C07326=1174.282,254.736,-65.728,-177.284,7.391,148.606
C07327=1174.278,254.984,-65.755,-177.282,7.393,148.606
C07328=1174.274,255.233,-65.782,-177.279,7.396,148.606
C07329=1174.270,255.482,-65.809,-177.276,7.399,148.606
C07330=1174.265,255.729,-65.836,-177.274,7.401,148.606
C07331=1174.261,255.978,-65.863,-177.272,7.404,148.606
C07332=1174.256,256.226,-65.890,-177.268,7.407,148.606
C07333=1174.252,256.475,-65.919,-177.266,7.409,148.605
C07334=1174.248,256.723,-65.946,-177.263,7.412,148.605
C07335=1174.243,256.971,-65.973,-177.261,7.415,148.605
C07336=1174.238,257.221,-66.001,-177.258,7.417,148.605
C07337=1174.234,257.469,-66.029,-177.256,7.420,148.605
C07338=1174.229,257.717,-66.056,-177.253,7.423,148.605
C07339=1174.225,257.966,-66.083,-177.250,7.425,148.605
C07340=1174.221,258.214,-66.111,-177.248,7.428,148.605
C07341=1174.216,258.463,-66.139,-177.245,7.431,148.605
C07342=1174.212,258.711,-66.166,-177.242,7.434,148.605
C07343=1174.208,258.960,-66.194,-177.240,7.436,148.605
C07344=1174.204,259.208,-66.222,-177.237,7.439,148.604
C07345=1174.199,259.456,-66.249,-177.234,7.441,148.604
C07346=1174.195,259.705,-66.277,-177.232,7.444,148.604
C07347=1174.191,259.953,-66.304,-177.229,7.447,148.604
C07348=1174.186,260.201,-66.332,-177.226,7.450,148.604
C07349=1174.181,260.451,-66.360,-177.224,7.452,148.604
C07350=1174.177,260.699,-66.387,-177.221,7.455,148.604
C07351=1174.172,260.947,-66.414,-177.219,7.458,148.604
C07352=1174.169,261.196,-66.443,-177.216,7.461,148.604
C07353=1174.164,261.443,-66.470,-177.213,7.462,148.603
C07354=1174.160,261.692,-66.497,-177.211,7.465,148.603
C07355=1174.155,261.965,-66.528,-177.208,7.468,148.603
C07356=1174.150,262.239,-66.559,-177.205,7.471,148.603
C07357=1174.145,262.511,-66.589,-177.202,7.474,148.603
C07358=1174.140,262.785,-66.620,-177.200,7.477,148.603
C07359=1174.136,263.032,-66.648,-177.196,7.480,148.603
C07360=1174.132,263.281,-66.676,-177.194,7.483,148.603
C07361=1174.127,263.529,-66.704,-177.191,7.486,148.603
C07362=1174.123,263.778,-66.731,-177.189,7.488,148.603
C07363=1174.119,264.026,-66.759,-177.186,7.491,148.603
C07364=1174.114,264.274,-66.788,-177.183,7.494,148.603
C07365=1174.110,264.523,-66.816,-177.180,7.497,148.603
C07366=1174.105,264.772,-66.843,-177.178,7.499,148.602
C07367=1174.102,265.020,-66.871,-177.176,7.502,148.602
C07368=1174.096,265.268,-66.899,-177.173,7.505,148.602
C07369=1174.093,265.517,-66.927,-177.171,7.507,148.602
C07370=1174.088,265.765,-66.955,-177.168,7.510,148.602
C07371=1174.083,266.014,-66.983,-177.165,7.513,148.602
C07372=1174.079,266.262,-67.011,-177.162,7.516,148.602
C07373=1174.075,266.510,-67.039,-177.160,7.518,148.602
C07374=1174.070,266.759,-67.068,-177.157,7.521,148.602
C07375=1174.066,267.007,-67.095,-177.154,7.524,148.602
C07376=1174.062,267.255,-67.124,-177.152,7.527,148.602
C07377=1174.057,267.504,-67.152,-177.149,7.529,148.602
C07378=1174.053,267.752,-67.180,-177.147,7.532,148.602
C07379=1174.048,268.000,-67.208,-177.144,7.535,148.602
C07380=1174.045,268.249,-67.237,-177.141,7.538,148.601
C07381=1174.040,268.497,-67.264,-177.139,7.540,148.601
C07382=1174.036,268.746,-67.293,-177.136,7.543,148.601
C07383=1174.031,268.994,-67.321,-177.133,7.546,148.601
C07384=1174.027,269.242,-67.350,-177.131,7.549,148.601
C07385=1174.023,269.490,-67.377,-177.128,7.552,148.601
C07386=1174.018,269.739,-67.406,-177.126,7.554,148.601
C07387=1174.014,269.987,-67.434,-177.123,7.557,148.601
C07388=1174.009,270.236,-67.463,-177.120,7.560,148.601
C07389=1174.005,270.484,-67.490,-177.118,7.563,148.601
C07390=1174.000,270.733,-67.519,-177.115,7.565,148.601
C07391=1173.997,270.981,-67.547,-177.113,7.568,148.601
C07392=1173.992,271.229,-67.575,-177.110,7.571,148.601
C07393=1173.988,271.478,-67.604,-177.107,7.574,148.601
C07394=1173.983,271.726,-67.633,-177.104,7.577,148.601
C07395=1173.979,271.974,-67.661,-177.102,7.579,148.601
C07396=1173.974,272.222,-67.689,-177.100,7.582,148.601
C07397=1173.970,272.471,-67.718,-177.097,7.585,148.601
C07398=1173.966,272.720,-67.746,-177.094,7.588,148.600
C07399=1173.962,272.968,-67.774,-177.092,7.590,148.600
C07400=1173.957,273.216,-67.803,-177.089,7.593,148.600
C07401=1173.953,273.464,-67.831,-177.086,7.596,148.600
C07402=1173.949,273.713,-67.860,-177.084,7.599,148.600
C07403=1173.944,273.962,-67.889,-177.081,7.602,148.600
C07404=1173.940,274.209,-67.917,-177.079,7.604,148.600
C07405=1173.936,274.458,-67.946,-177.076,7.607,148.600
C07406=1173.931,274.706,-67.974,-177.073,7.610,148.600
C07407=1173.927,274.954,-68.003,-177.071,7.613,148.600
C07408=1173.923,275.203,-68.032,-177.068,7.616,148.600
C07409=1173.918,275.451,-68.060,-177.066,7.618,148.600
C07410=1173.914,275.699,-68.089,-177.063,7.621,148.600
C07411=1173.910,275.948,-68.117,-177.060,7.624,148.600
C07412=1173.905,276.196,-68.146,-177.057,7.627,148.600
C07413=1173.901,276.444,-68.175,-177.055,7.630,148.600
C07414=1173.897,276.693,-68.203,-177.052,7.632,148.600
C07415=1173.892,276.940,-68.232,-177.050,7.635,148.600
C07416=1173.888,277.189,-68.261,-177.047,7.638,148.600
C07417=1173.884,277.438,-68.290,-177.044,7.641,148.599
C07418=1173.880,277.686,-68.319,-177.041,7.644,148.599
C07419=1173.875,277.934,-68.347,-177.039,7.647,148.599
C07420=1173.871,278.182,-68.377,-177.037,7.650,148.600
C07421=1173.867,278.431,-68.405,-177.034,7.653,148.599
C07422=1173.862,278.678,-68.434,-177.032,7.656,148.599
C07423=1173.858,278.927,-68.462,-177.029,7.659,148.599
C07424=1173.854,279.176,-68.492,-177.026,7.662,148.599
C07425=1173.850,279.424,-68.520,-177.024,7.664,148.599
C07426=1173.845,279.672,-68.549,-177.021,7.667,148.599
C07427=1173.841,279.920,-68.579,-177.018,7.670,148.599
C07428=1173.836,280.169,-68.607,-177.016,7.673,148.599
C07429=1173.832,280.417,-68.637,-177.013,7.676,148.599
C07430=1173.828,280.665,-68.665,-177.010,7.679,148.599
C07431=1173.824,280.913,-68.694,-177.008,7.681,148.599
C07432=1173.820,281.162,-68.723,-177.005,7.684,148.599
C07433=1173.815,281.410,-68.752,-177.003,7.687,148.599
C07434=1173.810,281.658,-68.781,-177.000,7.690,148.599
C07435=1173.806,281.906,-68.811,-176.998,7.693,148.599
C07436=1173.802,282.155,-68.840,-176.995,7.696,148.599
C07437=1173.798,282.403,-68.868,-176.992,7.699,148.599
C07438=1173.794,282.651,-68.898,-176.990,7.701,148.599
C07439=1173.789,282.900,-68.926,-176.987,7.704,148.599
C07440=1173.785,283.148,-68.956,-176.984,7.707,148.599
C07441=1173.780,283.396,-68.985,-176.982,7.710,148.599
C07442=1173.776,283.644,-69.015,-176.979,7.713,148.599
C07443=1173.772,283.893,-69.044,-176.977,7.716,148.599
C07444=1173.767,284.141,-69.072,-176.975,7.718,148.599
C07445=1173.763,284.389,-69.102,-176.972,7.721,148.599
C07446=1173.759,284.637,-69.131,-176.969,7.724,148.599
C07447=1173.754,284.886,-69.161,-176.966,7.727,148.599
C07448=1173.750,285.134,-69.190,-176.964,7.730,148.599
C07449=1173.746,285.383,-69.219,-176.961,7.733,148.599
C07450=1173.741,285.630,-69.248,-176.959,7.737,148.599
C07451=1173.737,285.879,-69.277,-176.956,7.739,148.599
C07452=1173.733,286.127,-69.307,-176.954,7.742,148.599
C07453=1173.728,286.375,-69.336,-176.951,7.745,148.599
C07454=1173.724,286.623,-69.366,-176.948,7.748,148.599
C07455=1173.720,286.872,-69.395,-176.945,7.751,148.599
C07456=1173.716,287.120,-69.425,-176.943,7.754,148.599
C07457=1173.712,287.368,-69.454,-176.940,7.757,148.599
C07458=1173.707,287.616,-69.483,-176.938,7.760,148.599
C07459=1173.702,287.891,-69.516,-176.935,7.763,148.599
C07460=1173.698,288.166,-69.549,-176.932,7.766,148.599
C07461=1173.693,288.441,-69.581,-176.929,7.769,148.599
C07462=1173.688,288.715,-69.614,-176.926,7.773,148.599
C07463=1173.684,288.963,-69.644,-176.923,7.776,148.599
C07464=1173.680,289.212,-69.673,-176.921,7.779,148.599
C07465=1173.675,289.460,-69.703,-176.919,7.781,148.599
C07466=1173.671,289.708,-69.732,-176.916,7.784,148.599
C07467=1173.667,289.956,-69.761,-176.913,7.787,148.599
C07468=1173.663,290.205,-69.791,-176.911,7.790,148.599
C07469=1173.659,290.453,-69.820,-176.908,7.793,148.599
C07470=1173.654,290.702,-69.850,-176.905,7.796,148.599
C07471=1173.650,290.949,-69.881,-176.903,7.799,148.599
C07472=1173.646,291.197,-69.910,-176.900,7.802,148.599
C07473=1173.642,291.446,-69.939,-176.898,7.805,148.599
C07474=1173.637,291.694,-69.969,-176.895,7.807,148.599
C07475=1173.632,291.943,-69.999,-176.893,7.810,148.599
C07476=1173.629,292.190,-70.029,-176.890,7.814,148.599
C07477=1173.624,292.438,-70.059,-176.888,7.817,148.599
C07478=1173.620,292.687,-70.088,-176.885,7.820,148.599
C07479=1173.616,292.935,-70.117,-176.882,7.823,148.599
C07480=1173.611,293.183,-70.148,-176.879,7.826,148.599
C07481=1173.607,293.431,-70.178,-176.877,7.829,148.599
C07482=1173.603,293.680,-70.207,-176.874,7.832,148.599
C07483=1173.599,293.928,-70.237,-176.872,7.835,148.599
C07484=1173.594,294.176,-70.267,-176.869,7.837,148.599
C07485=1173.590,294.424,-70.297,-176.867,7.840,148.599
C07486=1173.586,294.672,-70.326,-176.864,7.843,148.599
C07487=1173.582,294.920,-70.356,-176.862,7.846,148.599
C07488=1173.577,295.169,-70.386,-176.859,7.849,148.599
C07489=1173.573,295.416,-70.417,-176.857,7.853,148.599
C07490=1173.569,295.664,-70.446,-176.854,7.856,148.599
C07491=1173.564,295.913,-70.476,-176.851,7.859,148.599
C07492=1173.560,296.161,-70.506,-176.849,7.862,148.599
C07493=1173.557,296.410,-70.536,-176.846,7.865,148.599
C07494=1173.552,296.658,-70.567,-176.844,7.868,148.599
C07495=1173.548,296.906,-70.596,-176.841,7.871,148.599
C07496=1173.543,297.154,-70.627,-176.839,7.873,148.599
C07497=1173.539,297.402,-70.657,-176.836,7.876,148.599
C07498=1173.535,297.650,-70.687,-176.834,7.879,148.599
C07499=1173.530,297.898,-70.717,-176.831,7.882,148.599
C07500=1173.526,298.146,-70.747,-176.828,7.885,148.599
C07501=1173.521,298.395,-70.777,-176.826,7.888,148.599
C07502=1173.518,298.642,-70.807,-176.823,7.891,148.599
C07503=1173.514,298.891,-70.838,-176.820,7.894,148.599
C07504=1173.509,299.139,-70.868,-176.818,7.897,148.599
C07505=1173.506,299.387,-70.898,-176.815,7.901,148.599
C07506=1173.501,299.635,-70.928,-176.813,7.904,148.599
C07507=1173.497,299.883,-70.958,-176.810,7.907,148.599
C07508=1173.492,300.131,-70.989,-176.807,7.910,148.599
C07509=1173.489,300.380,-71.019,-176.805,7.913,148.599
C07510=1173.484,300.628,-71.050,-176.802,7.916,148.599
C07511=1173.480,300.875,-71.080,-176.800,7.918,148.599
C07512=1173.475,301.124,-71.110,-176.798,7.921,148.600
C07513=1173.471,301.372,-71.140,-176.795,7.924,148.599
C07514=1173.467,301.620,-71.171,-176.792,7.927,148.599
C07515=1173.463,301.869,-71.200,-176.790,7.931,148.600
C07516=1173.458,302.117,-71.231,-176.787,7.934,148.600
C07517=1173.455,302.364,-71.261,-176.785,7.937,148.600
C07518=1173.450,302.612,-71.292,-176.782,7.940,148.600
C07519=1173.445,302.860,-71.323,-176.779,7.943,148.600
C07520=1173.442,303.109,-71.353,-176.777,7.946,148.600
C07521=1173.437,303.357,-71.384,-176.774,7.949,148.600
C07522=1173.433,303.605,-71.414,-176.772,7.952,148.600
C07523=1173.429,303.853,-71.444,-176.769,7.955,148.600
C07524=1173.424,304.101,-71.475,-176.766,7.958,148.600
C07525=1173.421,304.349,-71.506,-176.764,7.961,148.600
C07526=1173.416,304.598,-71.536,-176.761,7.964,148.600
C07527=1173.411,304.846,-71.567,-176.759,7.967,148.600
C07528=1173.407,305.093,-71.597,-176.756,7.971,148.600
C07529=1173.403,305.342,-71.628,-176.754,7.974,148.600
C07530=1173.399,305.590,-71.659,-176.751,7.977,148.600
C07531=1173.395,305.837,-71.689,-176.749,7.980,148.600
C07532=1173.391,306.086,-71.720,-176.746,7.983,148.600
C07533=1173.386,306.334,-71.751,-176.744,7.986,148.601
C07534=1173.382,306.582,-71.781,-176.741,7.988,148.600
C07535=1173.378,306.830,-71.812,-176.739,7.991,148.600
C07536=1173.374,307.078,-71.843,-176.736,7.995,148.601
C07537=1173.369,307.326,-71.874,-176.734,7.998,148.601
C07538=1173.365,307.574,-71.904,-176.731,8.001,148.601
C07539=1173.361,307.823,-71.935,-176.729,8.004,148.601
C07540=1173.357,308.071,-71.966,-176.726,8.007,148.601
C07541=1173.352,308.319,-71.996,-176.723,8.010,148.601
C07542=1173.349,308.567,-72.027,-176.721,8.013,148.601
C07543=1173.344,308.815,-72.058,-176.718,8.016,148.601
C07544=1173.340,309.062,-72.089,-176.716,8.020,148.601
C07545=1173.336,309.311,-72.120,-176.713,8.023,148.601
C07546=1173.331,309.559,-72.151,-176.710,8.025,148.601
C07547=1173.327,309.806,-72.181,-176.708,8.029,148.601
C07548=1173.323,310.055,-72.212,-176.705,8.032,148.601
C07549=1173.319,310.303,-72.243,-176.703,8.035,148.601
C07550=1173.314,310.550,-72.275,-176.700,8.038,148.601
C07551=1173.310,310.799,-72.306,-176.698,8.041,148.601
C07552=1173.306,311.047,-72.336,-176.695,8.044,148.602
C07553=1173.302,311.295,-72.367,-176.693,8.047,148.602
C07554=1173.298,311.543,-72.398,-176.690,8.051,148.602
C07555=1173.294,311.791,-72.429,-176.688,8.054,148.602
C07556=1173.290,312.039,-72.460,-176.685,8.057,148.602
C07557=1173.285,312.287,-72.491,-176.683,8.060,148.602
C07558=1173.281,312.535,-72.523,-176.680,8.063,148.602
C07559=1173.277,312.783,-72.554,-176.678,8.066,148.602
C07560=1173.272,313.031,-72.584,-176.675,8.069,148.602
C07561=1173.268,313.279,-72.616,-176.673,8.072,148.602
C07562=1173.264,313.527,-72.647,-176.670,8.075,148.602
C07563=1173.260,313.804,-72.682,-176.667,8.079,148.602
C07564=1173.254,314.081,-72.716,-176.664,8.083,148.602
C07565=1173.250,314.358,-72.751,-176.661,8.086,148.603
C07566=1173.245,314.634,-72.786,-176.659,8.090,148.603
C07567=1173.241,314.883,-72.817,-176.656,8.093,148.603
C07568=1173.237,315.130,-72.849,-176.653,8.096,148.603
C07569=1173.233,315.379,-72.880,-176.651,8.099,148.603
C07570=1173.229,315.626,-72.911,-176.648,8.102,148.603
C07571=1173.225,315.875,-72.943,-176.646,8.105,148.603
C07572=1173.220,316.122,-72.974,-176.643,8.108,148.603
C07573=1173.216,316.371,-73.005,-176.641,8.112,148.603
C07574=1173.212,316.618,-73.037,-176.638,8.115,148.603
C07575=1173.208,316.867,-73.068,-176.636,8.118,148.603
C07576=1173.204,317.114,-73.099,-176.633,8.121,148.603
C07577=1173.200,317.362,-73.131,-176.631,8.124,148.604
C07578=1173.195,317.610,-73.162,-176.628,8.127,148.604
C07579=1173.192,317.858,-73.194,-176.626,8.130,148.604
C07580=1173.187,318.106,-73.224,-176.623,8.133,148.604
C07581=1173.183,318.355,-73.257,-176.621,8.137,148.604
C07582=1173.178,318.602,-73.288,-176.618,8.140,148.604
C07583=1173.174,318.851,-73.319,-176.616,8.143,148.604
C07584=1173.170,319.099,-73.351,-176.613,8.147,148.604
C07585=1173.166,319.346,-73.383,-176.610,8.150,148.604
C07586=1173.162,319.595,-73.414,-176.608,8.153,148.604
C07587=1173.158,319.842,-73.445,-176.605,8.156,148.605
C07588=1173.153,320.091,-73.478,-176.603,8.159,148.605
C07589=1173.149,320.338,-73.509,-176.600,8.163,148.605
C07590=1173.145,320.587,-73.540,-176.598,8.166,148.605
C07591=1173.141,320.835,-73.572,-176.595,8.169,148.605
C07592=1173.137,321.082,-73.604,-176.593,8.172,148.605
C07593=1173.133,321.330,-73.636,-176.590,8.175,148.605
C07594=1173.128,321.578,-73.667,-176.588,8.178,148.605
C07595=1173.124,321.826,-73.699,-176.585,8.182,148.605
C07596=1173.121,322.074,-73.731,-176.583,8.185,148.606
C07597=1173.116,322.322,-73.762,-176.580,8.188,148.606
C07598=1173.112,322.570,-73.795,-176.578,8.191,148.606
C07599=1173.108,322.818,-73.826,-176.575,8.194,148.606
C07600=1173.104,323.066,-73.857,-176.573,8.197,148.606
C07601=1173.100,323.314,-73.889,-176.570,8.200,148.606
C07602=1173.095,323.562,-73.921,-176.568,8.204,148.606
C07603=1173.091,323.810,-73.953,-176.566,8.207,148.606
C07604=1173.087,324.058,-73.985,-176.563,8.210,148.606
C07605=1173.084,324.306,-74.017,-176.560,8.214,148.607
C07606=1173.079,324.553,-74.049,-176.557,8.217,148.607
C07607=1173.075,324.801,-74.081,-176.555,8.220,148.607
C07608=1173.071,325.049,-74.112,-176.552,8.223,148.607
C07609=1173.066,325.297,-74.145,-176.550,8.227,148.607
C07610=1173.062,325.545,-74.176,-176.548,8.230,148.607
C07611=1173.059,325.793,-74.208,-176.545,8.233,148.607
C07612=1173.054,326.041,-74.240,-176.543,8.236,148.607
C07613=1173.050,326.289,-74.272,-176.541,8.240,148.608
C07614=1173.046,326.537,-74.305,-176.538,8.243,148.608
C07615=1173.041,326.785,-74.336,-176.536,8.246,148.608
C07616=1173.038,327.033,-74.368,-176.533,8.249,148.608
C07617=1173.033,327.281,-74.400,-176.531,8.252,148.608
C07618=1173.030,327.528,-74.433,-176.528,8.255,148.608
C07619=1173.025,327.776,-74.465,-176.526,8.258,148.608
C07620=1173.021,328.024,-74.497,-176.523,8.263,148.608
C07621=1173.017,328.272,-74.529,-176.520,8.266,148.609
C07622=1173.013,328.520,-74.561,-176.518,8.269,148.609
C07623=1173.008,328.768,-74.593,-176.515,8.272,148.609
C07624=1173.004,329.016,-74.626,-176.513,8.275,148.609
C07625=1173.001,329.264,-74.658,-176.510,8.278,148.609
C07626=1172.996,329.512,-74.690,-176.508,8.282,148.609
C07627=1172.992,329.759,-74.721,-176.506,8.285,148.609
C07628=1172.988,330.007,-74.755,-176.503,8.288,148.609
C07629=1172.984,330.255,-74.786,-176.501,8.291,148.610
C07630=1172.980,330.503,-74.819,-176.499,8.295,148.610
C07631=1172.975,330.751,-74.850,-176.496,8.298,148.610
C07632=1172.971,330.998,-74.884,-176.493,8.302,148.610
C07633=1172.967,331.246,-74.915,-176.491,8.305,148.610
C07634=1172.963,331.495,-74.948,-176.488,8.308,148.610
C07635=1172.959,331.743,-74.981,-176.486,8.311,148.610
C07636=1172.955,331.990,-75.012,-176.483,8.315,148.611
C07637=1172.950,332.238,-75.045,-176.481,8.318,148.611
C07638=1172.947,332.486,-75.077,-176.478,8.321,148.611
C07639=1172.942,332.734,-75.110,-176.476,8.324,148.611
C07640=1172.938,332.982,-75.143,-176.474,8.328,148.611
C07641=1172.934,333.230,-75.175,-176.471,8.331,148.611
C07642=1172.930,333.478,-75.208,-176.468,8.335,148.612
C07643=1172.926,333.725,-75.240,-176.466,8.338,148.612
C07644=1172.922,333.973,-75.273,-176.464,8.341,148.612
C07645=1172.917,334.221,-75.305,-176.461,8.344,148.612
C07646=1172.914,334.468,-75.338,-176.459,8.348,148.612
C07647=1172.910,334.717,-75.370,-176.456,8.351,148.612
C07648=1172.905,334.964,-75.403,-176.454,8.354,148.613
C07649=1172.902,335.212,-75.435,-176.451,8.357,148.613
C07650=1172.897,335.459,-75.468,-176.449,8.360,148.613
C07651=1172.893,335.708,-75.500,-176.446,8.365,148.613
C07652=1172.889,335.955,-75.533,-176.444,8.368,148.613
C07653=1172.885,336.204,-75.565,-176.442,8.371,148.613
C07654=1172.881,336.451,-75.599,-176.439,8.374,148.613
C07655=1172.876,336.699,-75.632,-176.437,8.377,148.614
C07656=1172.873,336.947,-75.664,-176.434,8.381,148.614
C07657=1172.869,337.195,-75.697,-176.432,8.384,148.614
C07658=1172.864,337.443,-75.730,-176.430,8.387,148.614
C07659=1172.860,337.691,-75.762,-176.427,8.391,148.614
C07660=1172.857,337.938,-75.795,-176.424,8.394,148.615
C07661=1172.852,338.186,-75.828,-176.422,8.398,148.615
C07662=1172.848,338.434,-75.860,-176.420,8.401,148.615
C07663=1172.844,338.682,-75.894,-176.418,8.404,148.615
C07664=1172.840,338.930,-75.927,-176.415,8.408,148.615
C07665=1172.836,339.177,-75.959,-176.413,8.411,148.615
C07666=1172.831,339.425,-75.991,-176.410,8.415,148.616
C07667=1172.827,339.705,-76.029,-176.407,8.418,148.616
C07668=1172.822,339.984,-76.066,-176.405,8.422,148.616
C07669=1172.818,340.263,-76.103,-176.402,8.426,148.616
C07670=1172.813,340.542,-76.141,-176.399,8.430,148.617
C07671=1172.809,340.790,-76.174,-176.397,8.433,148.617
C07672=1172.805,341.038,-76.207,-176.394,8.436,148.617
C07673=1172.800,341.286,-76.239,-176.392,8.440,148.617
C07674=1172.796,341.534,-76.272,-176.389,8.443,148.617
C07675=1172.793,341.781,-76.305,-176.387,8.447,148.617
C07676=1172.789,342.029,-76.338,-176.385,8.450,148.618
C07677=1172.784,342.277,-76.371,-176.382,8.453,148.618
C07678=1172.780,342.524,-76.405,-176.380,8.457,148.618
C07679=1172.776,342.772,-76.438,-176.377,8.461,148.618
C07680=1172.772,343.020,-76.471,-176.375,8.464,148.619
C07681=1172.768,343.268,-76.504,-176.373,8.467,148.619
C07682=1172.764,343.515,-76.537,-176.370,8.471,148.619
C07683=1172.760,343.763,-76.570,-176.368,8.474,148.619
C07684=1172.756,344.011,-76.603,-176.366,8.477,148.619
C07685=1172.751,344.258,-76.637,-176.363,8.481,148.620
C07686=1172.747,344.506,-76.670,-176.360,8.484,148.620
C07687=1172.743,344.754,-76.703,-176.358,8.488,148.620
C07688=1172.740,345.002,-76.736,-176.356,8.491,148.620
C07689=1172.735,345.250,-76.770,-176.354,8.494,148.620
C07690=1172.731,345.498,-76.803,-176.351,8.498,148.621
C07691=1172.727,345.746,-76.836,-176.348,8.502,148.621
C07692=1172.723,345.993,-76.870,-176.346,8.505,148.621
C07693=1172.719,346.240,-76.903,-176.344,8.508,148.621
C07694=1172.714,346.488,-76.937,-176.342,8.512,148.621
C07695=1172.710,346.736,-76.970,-176.339,8.515,148.622
C07696=1172.706,346.984,-77.003,-176.337,8.519,148.622
C07697=1172.702,347.232,-77.036,-176.335,8.523,148.622
C07698=1172.699,347.479,-77.070,-176.332,8.526,148.623
C07699=1172.695,347.727,-77.104,-176.330,8.529,148.623
C07700=1172.690,347.975,-77.137,-176.328,8.533,148.623
C07701=1172.686,348.223,-77.170,-176.325,8.536,148.623
C07702=1172.682,348.470,-77.204,-176.323,8.540,148.623
C07703=1172.678,348.718,-77.237,-176.320,8.543,148.624
C07704=1172.674,348.966,-77.271,-176.318,8.547,148.624
C07705=1172.670,349.213,-77.305,-176.316,8.550,148.624
C07706=1172.666,349.461,-77.338,-176.313,8.553,148.624
C07707=1172.662,349.709,-77.371,-176.311,8.557,148.625
C07708=1172.658,349.956,-77.405,-176.308,8.561,148.625
C07709=1172.653,350.204,-77.439,-176.306,8.564,148.625
C07710=1172.650,350.452,-77.472,-176.304,8.568,148.625
C07711=1172.646,350.699,-77.506,-176.302,8.571,148.626
C07712=1172.642,350.947,-77.539,-176.299,8.575,148.626
C07713=1172.637,351.195,-77.573,-176.297,8.578,148.626
C07714=1172.633,351.442,-77.607,-176.295,8.582,148.626
C07715=1172.629,351.691,-77.640,-176.292,8.585,148.627
C07716=1172.626,351.938,-77.674,-176.290,8.588,148.627
C07717=1172.621,352.186,-77.708,-176.288,8.593,148.627
C07718=1172.617,352.433,-77.742,-176.285,8.596,148.627
C07719=1172.613,352.681,-77.776,-176.283,8.599,148.628
C07720=1172.610,352.929,-77.809,-176.281,8.603,148.628
C07721=1172.605,353.177,-77.843,-176.278,8.607,148.628
C07722=1172.601,353.424,-77.877,-176.276,8.610,148.629
C07723=1172.597,353.672,-77.911,-176.274,8.614,148.629
C07724=1172.593,353.920,-77.945,-176.271,8.617,148.629
C07725=1172.589,354.167,-77.979,-176.269,8.620,148.629
C07726=1172.585,354.414,-78.012,-176.267,8.625,148.630
C07727=1172.581,354.663,-78.047,-176.265,8.628,148.630
C07728=1172.577,354.910,-78.080,-176.262,8.631,148.630
C07729=1172.573,355.157,-78.114,-176.260,8.634,148.630
C07730=1172.569,355.405,-78.149,-176.258,8.639,148.631
C07731=1172.565,355.653,-78.182,-176.255,8.642,148.631
C07732=1172.560,355.901,-78.216,-176.253,8.646,148.631
C07733=1172.557,356.148,-78.251,-176.251,8.649,148.632
C07734=1172.553,356.396,-78.284,-176.248,8.653,148.632
C07735=1172.548,356.644,-78.318,-176.246,8.657,148.632
C07736=1172.545,356.891,-78.352,-176.244,8.660,148.632
C07737=1172.540,357.139,-78.387,-176.242,8.663,148.633
C07738=1172.536,357.387,-78.420,-176.239,8.668,148.633
C07739=1172.533,357.634,-78.454,-176.237,8.671,148.633
C07740=1172.528,357.882,-78.489,-176.235,8.675,148.634
C07741=1172.525,358.129,-78.523,-176.233,8.678,148.634
C07742=1172.520,358.378,-78.557,-176.230,8.682,148.634
C07743=1172.517,358.625,-78.591,-176.228,8.686,148.635
C07744=1172.512,358.872,-78.625,-176.226,8.689,148.635
C07745=1172.509,359.120,-78.659,-176.224,8.692,148.635
C07746=1172.504,359.367,-78.694,-176.221,8.697,148.636
C07747=1172.501,359.615,-78.728,-176.219,8.700,148.636
C07748=1172.496,359.863,-78.762,-176.217,8.704,148.636
C07749=1172.493,360.110,-78.796,-176.215,8.707,148.637
C07750=1172.488,360.358,-78.830,-176.212,8.711,148.637
C07751=1172.484,360.606,-78.864,-176.210,8.715,148.637
C07752=1172.480,360.854,-78.899,-176.208,8.718,148.638
C07753=1172.477,361.101,-78.933,-176.206,8.721,148.638
C07754=1172.472,361.348,-78.968,-176.203,8.726,148.638
C07755=1172.468,361.596,-79.002,-176.202,8.730,148.639
C07756=1172.464,361.843,-79.036,-176.199,8.733,148.639
C07757=1172.460,362.092,-79.071,-176.197,8.736,148.639
C07758=1172.456,362.339,-79.105,-176.195,8.741,148.640
C07759=1172.452,362.587,-79.140,-176.193,8.744,148.640
C07760=1172.448,362.834,-79.174,-176.191,8.748,148.641
C07761=1172.445,363.081,-79.209,-176.189,8.751,148.641
C07762=1172.440,363.329,-79.244,-176.187,8.755,148.641
C07763=1172.437,363.577,-79.278,-176.184,8.759,148.642
C07764=1172.433,363.824,-79.312,-176.182,8.762,148.642
C07765=1172.429,364.072,-79.347,-176.180,8.766,148.642
C07766=1172.425,364.319,-79.381,-176.178,8.770,148.643
C07767=1172.421,364.567,-79.416,-176.176,8.773,148.643
C07768=1172.416,364.815,-79.450,-176.174,8.777,148.643
C07769=1172.413,365.062,-79.485,-176.172,8.781,148.644
C07770=1172.409,365.309,-79.520,-176.170,8.785,148.644
C07771=1172.404,365.592,-79.560,-176.168,8.789,148.645
C07772=1172.399,365.874,-79.598,-176.166,8.793,148.645
C07773=1172.395,366.156,-79.638,-176.163,8.797,148.646
C07774=1172.390,366.438,-79.678,-176.161,8.801,148.646
C07775=1172.387,366.685,-79.713,-176.159,8.805,148.647
C07776=1172.383,366.933,-79.747,-176.157,8.809,148.647
C07777=1172.379,367.181,-79.782,-176.155,8.812,148.647
C07778=1172.374,367.428,-79.816,-176.154,8.816,148.648
C07779=1172.371,367.675,-79.851,-176.152,8.820,148.648
C07780=1172.367,367.923,-79.886,-176.150,8.823,148.649
C07781=1172.363,368.171,-79.921,-176.147,8.828,148.649
C07782=1172.358,368.418,-79.956,-176.146,8.831,148.650
C07783=1172.354,368.666,-79.991,-176.144,8.835,148.650
C07784=1172.351,368.913,-80.024,-176.142,8.838,148.651
C07785=1172.347,369.160,-80.060,-176.140,8.842,148.651
C07786=1172.343,369.409,-80.095,-176.139,8.846,148.652
C07787=1172.339,369.655,-80.130,-176.137,8.850,148.652
C07788=1172.335,369.904,-80.165,-176.135,8.853,148.652
C07789=1172.330,370.151,-80.199,-176.133,8.857,148.653
C07790=1172.326,370.398,-80.235,-176.132,8.861,148.653
C07791=1172.323,370.646,-80.269,-176.130,8.864,148.654
C07792=1172.319,370.893,-80.304,-176.128,8.868,148.654
C07793=1172.315,371.141,-80.339,-176.127,8.872,148.655
C07794=1172.311,371.388,-80.374,-176.125,8.875,148.655
C07795=1172.307,371.636,-80.409,-176.123,8.879,148.656
C07796=1172.303,371.884,-80.445,-176.122,8.883,148.656
C07797=1172.299,372.131,-80.479,-176.120,8.886,148.657
C07798=1172.295,372.378,-80.515,-176.119,8.890,148.657
C07799=1172.291,372.627,-80.550,-176.117,8.893,148.658
C07800=1172.287,372.873,-80.585,-176.116,8.897,148.659
C07801=1172.284,373.121,-80.620,-176.114,8.901,148.659
C07802=1172.279,373.368,-80.654,-176.112,8.905,148.660
C07803=1172.276,373.616,-80.690,-176.111,8.908,148.660
C07804=1172.272,373.864,-80.724,-176.110,8.911,148.661
C07805=1172.267,374.110,-80.760,-176.108,8.915,148.661
C07806=1172.264,374.358,-80.795,-176.106,8.919,148.662
C07807=1172.260,374.606,-80.830,-176.105,8.923,148.662
C07808=1172.255,374.853,-80.865,-176.104,8.927,148.663
C07809=1172.252,375.100,-80.901,-176.102,8.929,148.663
C07810=1172.248,375.348,-80.936,-176.101,8.933,148.664
C07811=1172.244,375.596,-80.971,-176.100,8.937,148.665
C07812=1172.240,375.843,-81.006,-176.099,8.940,148.665
C07813=1172.236,376.091,-81.041,-176.097,8.944,148.666
C07814=1172.232,376.338,-81.077,-176.095,8.948,148.666
C07815=1172.228,376.585,-81.112,-176.095,8.951,148.667
C07816=1172.224,376.833,-81.147,-176.093,8.955,148.667
C07817=1172.220,377.081,-81.182,-176.092,8.959,148.668
C07818=1172.216,377.328,-81.217,-176.091,8.962,148.669
C07819=1172.212,377.575,-81.254,-176.090,8.966,148.669
C07820=1172.208,377.823,-81.289,-176.089,8.969,148.670
C07821=1172.204,378.071,-81.324,-176.087,8.973,148.670
C07822=1172.200,378.318,-81.359,-176.086,8.976,148.671
C07823=1172.196,378.565,-81.395,-176.085,8.980,148.672
C07824=1172.192,378.813,-81.430,-176.084,8.984,148.672
C07825=1172.188,379.060,-81.465,-176.083,8.987,148.673
C07826=1172.184,379.308,-81.500,-176.082,8.990,148.673
C07827=1172.181,379.555,-81.536,-176.081,8.994,148.674
C07828=1172.177,379.803,-81.571,-176.080,8.997,148.675
C07829=1172.172,380.050,-81.607,-176.079,9.001,148.675
C07830=1172.168,380.297,-81.643,-176.078,9.004,148.676
C07831=1172.165,380.545,-81.678,-176.077,9.007,148.677
C07832=1172.161,380.792,-81.714,-176.076,9.012,148.677
C07833=1172.156,381.040,-81.748,-176.075,9.015,148.678
C07834=1172.153,381.287,-81.784,-176.074,9.018,148.679
C07835=1172.149,381.535,-81.819,-176.073,9.022,148.679
C07836=1172.145,381.783,-81.856,-176.073,9.025,148.680
C07837=1172.141,382.030,-81.891,-176.072,9.028,148.681
C07838=1172.137,382.277,-81.926,-176.071,9.032,148.681
C07839=1172.133,382.524,-81.962,-176.070,9.035,148.682
C07840=1172.129,382.772,-81.997,-176.069,9.039,148.683
C07841=1172.126,383.019,-82.033,-176.069,9.042,148.683
C07842=1172.121,383.267,-82.069,-176.068,9.045,148.684
C07843=1172.117,383.514,-82.104,-176.067,9.048,148.685
C07844=1172.113,383.762,-82.140,-176.067,9.051,148.685
C07845=1172.110,384.009,-82.175,-176.066,9.055,148.686
C07846=1172.106,384.257,-82.211,-176.065,9.058,148.687
C07847=1172.101,384.504,-82.247,-176.064,9.062,148.687
C07848=1172.097,384.751,-82.282,-176.063,9.065,148.688
C07849=1172.094,384.999,-82.318,-176.063,9.069,148.689
C07850=1172.090,385.246,-82.353,-176.063,9.071,148.690
C07851=1172.086,385.494,-82.389,-176.062,9.074,148.690
C07852=1172.082,385.741,-82.425,-176.062,9.078,148.691
C07853=1172.078,385.988,-82.460,-176.061,9.081,148.691
C07854=1172.074,386.236,-82.496,-176.061,9.084,148.692
C07855=1172.070,386.484,-82.532,-176.060,9.088,148.693
C07856=1172.066,386.730,-82.568,-176.059,9.091,148.694
C07857=1172.063,386.978,-82.604,-176.060,9.093,148.694
C07858=1172.059,387.225,-82.639,-176.059,9.097,148.695
C07859=1172.054,387.473,-82.675,-176.059,9.100,148.696
C07860=1172.050,387.720,-82.711,-176.058,9.103,148.696
C07861=1172.047,387.968,-82.746,-176.058,9.106,148.697
C07862=1172.043,388.215,-82.782,-176.058,9.109,148.698
C07863=1172.039,388.463,-82.818,-176.057,9.112,148.699
C07864=1172.035,388.710,-82.854,-176.057,9.115,148.699
C07865=1172.031,388.957,-82.889,-176.057,9.118,148.700
C07866=1172.027,389.204,-82.925,-176.057,9.121,148.701
C07867=1172.023,389.452,-82.961,-176.056,9.124,148.701
C07868=1172.019,389.699,-82.996,-176.056,9.127,148.702
C07869=1172.015,389.947,-83.033,-176.056,9.130,148.703
C07870=1172.011,390.194,-83.069,-176.056,9.133,148.704
C07871=1172.008,390.442,-83.104,-176.056,9.136,148.704
C07872=1172.004,390.689,-83.140,-176.056,9.139,148.705
C07873=1171.999,390.936,-83.176,-176.056,9.142,148.706
C07874=1171.995,391.184,-83.211,-176.055,9.144,148.706
C07875=1171.991,391.468,-83.253,-176.055,9.148,148.707
C07876=1171.986,391.753,-83.294,-176.055,9.151,148.708
C07877=1171.983,392.038,-83.336,-176.055,9.154,148.709
C07878=1171.978,392.323,-83.377,-176.055,9.158,148.710
C07879=1171.974,392.571,-83.413,-176.055,9.160,148.711
C07880=1171.970,392.817,-83.449,-176.055,9.163,148.711
C07881=1171.966,393.064,-83.484,-176.055,9.166,148.712
C07882=1171.962,393.312,-83.520,-176.055,9.169,148.713
C07883=1171.958,393.560,-83.556,-176.055,9.171,148.714
C07884=1171.955,393.807,-83.592,-176.055,9.174,148.714
C07885=1171.950,394.054,-83.628,-176.055,9.176,148.715
C07886=1171.946,394.302,-83.664,-176.055,9.179,148.715
C07887=1171.943,394.549,-83.699,-176.055,9.181,148.716
C07888=1171.939,394.797,-83.736,-176.055,9.185,148.717
C07889=1171.935,395.044,-83.772,-176.055,9.187,148.718
C07890=1171.930,395.291,-83.808,-176.055,9.190,148.718
C07891=1171.927,395.538,-83.844,-176.056,9.192,148.719
C07892=1171.923,395.786,-83.879,-176.056,9.195,148.720
C07893=1171.919,396.033,-83.915,-176.056,9.197,148.721
C07894=1171.915,396.281,-83.951,-176.056,9.200,148.721
C07895=1171.911,396.528,-83.988,-176.056,9.203,148.722
C07896=1171.907,396.776,-84.023,-176.056,9.205,148.723
C07897=1171.904,397.023,-84.059,-176.056,9.208,148.723
C07898=1171.899,397.270,-84.096,-176.057,9.210,148.724
C07899=1171.896,397.518,-84.131,-176.057,9.212,148.725
C07900=1171.891,397.766,-84.168,-176.057,9.215,148.725
C07901=1171.887,398.012,-84.203,-176.058,9.217,148.726
C07902=1171.884,398.259,-84.239,-176.057,9.219,148.727
C07903=1171.879,398.507,-84.275,-176.057,9.222,148.727
C07904=1171.876,398.754,-84.311,-176.058,9.225,148.728
C07905=1171.872,399.002,-84.348,-176.058,9.227,148.729
C07906=1171.868,399.249,-84.383,-176.059,9.229,148.729
C07907=1171.864,399.496,-84.420,-176.059,9.231,148.730
C07908=1171.860,399.744,-84.455,-176.059,9.234,148.731
C07909=1171.857,399.991,-84.492,-176.059,9.237,148.732
C07910=1171.852,400.239,-84.528,-176.060,9.238,148.732
C07911=1171.849,400.486,-84.563,-176.060,9.241,148.733
C07912=1171.845,400.733,-84.600,-176.060,9.243,148.734
C07913=1171.841,400.981,-84.636,-176.060,9.246,148.734
C07914=1171.836,401.228,-84.672,-176.060,9.247,148.735
C07915=1171.833,401.475,-84.708,-176.061,9.250,148.736
C07916=1171.828,401.723,-84.744,-176.061,9.253,148.736
C07917=1171.825,401.970,-84.780,-176.061,9.254,148.737
C07918=1171.821,402.217,-84.816,-176.061,9.257,148.737
C07919=1171.817,402.465,-84.852,-176.061,9.259,148.738
C07920=1171.813,402.712,-84.888,-176.062,9.261,148.739
C07921=1171.809,402.960,-84.924,-176.062,9.263,148.740
C07922=1171.806,403.206,-84.961,-176.062,9.266,148.740
C07923=1171.801,403.454,-84.997,-176.063,9.267,148.741
C07924=1171.798,403.702,-85.032,-176.063,9.270,148.741
C07925=1171.794,403.949,-85.069,-176.063,9.272,148.742
C07926=1171.790,404.196,-85.105,-176.064,9.274,148.743
C07927=1171.786,404.444,-85.142,-176.064,9.276,148.743
C07928=1171.782,404.691,-85.177,-176.064,9.278,148.744
C07929=1171.778,404.939,-85.213,-176.065,9.280,148.745
C07930=1171.774,405.186,-85.250,-176.065,9.283,148.745
C07931=1171.771,405.433,-85.285,-176.065,9.285,148.746
C07932=1171.766,405.680,-85.322,-176.065,9.287,148.747
C07933=1171.762,405.927,-85.357,-176.066,9.289,148.747
C07934=1171.758,406.174,-85.394,-176.066,9.291,148.748
C07935=1171.755,406.422,-85.430,-176.066,9.293,148.748
C07936=1171.750,406.670,-85.466,-176.067,9.295,148.749
C07937=1171.747,406.917,-85.502,-176.067,9.297,148.750
C07938=1171.742,407.164,-85.538,-176.067,9.299,148.750
C07939=1171.739,407.411,-85.574,-176.068,9.301,148.751
C07940=1171.735,407.659,-85.611,-176.068,9.303,148.751
C07941=1171.731,407.906,-85.647,-176.068,9.305,148.752
C07942=1171.727,408.154,-85.683,-176.068,9.307,148.753
C07943=1171.724,408.401,-85.719,-176.069,9.309,148.753
C07944=1171.719,408.649,-85.755,-176.069,9.311,148.754
C07945=1171.716,408.895,-85.792,-176.069,9.313,148.754
C07946=1171.711,409.143,-85.828,-176.070,9.315,148.755
C07947=1171.708,409.390,-85.864,-176.070,9.317,148.756
C07948=1171.704,409.638,-85.900,-176.070,9.319,148.756
C07949=1171.700,409.885,-85.936,-176.070,9.321,148.757
C07950=1171.696,410.133,-85.973,-176.071,9.323,148.757
C07951=1171.693,410.379,-86.009,-176.071,9.324,148.758
C07952=1171.688,410.627,-86.045,-176.071,9.327,148.759
C07953=1171.685,410.874,-86.081,-176.072,9.328,148.759
C07954=1171.680,411.122,-86.117,-176.072,9.330,148.760
C07955=1171.677,411.370,-86.153,-176.072,9.332,148.760
C07956=1171.673,411.617,-86.190,-176.073,9.334,148.761
C07957=1171.669,411.864,-86.225,-176.073,9.336,148.762
C07958=1171.665,412.111,-86.262,-176.073,9.338,148.762
C07959=1171.661,412.359,-86.298,-176.074,9.339,148.763
C07960=1171.657,412.606,-86.335,-176.073,9.342,148.763
C07961=1171.654,412.853,-86.371,-176.074,9.343,148.764
C07962=1171.649,413.101,-86.407,-176.074,9.345,148.764
C07963=1171.646,413.348,-86.443,-176.074,9.347,148.765
C07964=1171.642,413.595,-86.479,-176.075,9.349,148.765
C07965=1171.638,413.842,-86.516,-176.075,9.350,148.766
C07966=1171.634,414.090,-86.552,-176.075,9.353,148.767
C07967=1171.630,414.337,-86.588,-176.076,9.354,148.767
C07968=1171.626,414.585,-86.624,-176.076,9.356,148.767
C07969=1171.621,414.831,-86.661,-176.077,9.358,148.768
C07970=1171.618,415.079,-86.696,-176.076,9.360,148.769
C07971=1171.614,415.327,-86.733,-176.077,9.362,148.769
C07972=1171.611,415.574,-86.769,-176.077,9.363,148.770
C07973=1171.609,415.821,-86.805,-176.077,9.365,148.770
C07974=1171.607,416.069,-86.841,-176.077,9.367,148.771
C07975=1171.606,416.344,-86.881,-176.078,9.368,148.771
C07976=1171.607,416.619,-86.921,-176.078,9.371,148.772
C07977=1171.609,416.895,-86.961,-176.078,9.372,148.772
C07978=1171.612,417.169,-87.000,-176.079,9.374,148.773
C07979=1171.191,417.170,-87.045,-176.082,9.385,148.777
C07980=1171.188,416.892,-87.005,-176.081,9.383,148.776
C07981=1171.185,416.614,-86.965,-176.081,9.382,148.776
C07982=1171.185,416.336,-86.924,-176.081,9.379,148.775
C07983=1171.185,416.057,-86.884,-176.081,9.378,148.775
C07984=1171.187,415.810,-86.847,-176.080,9.376,148.774
C07985=1171.189,415.563,-86.811,-176.080,9.374,148.773
C07986=1171.193,415.315,-86.776,-176.080,9.372,148.773
C07987=1171.197,415.068,-86.739,-176.080,9.371,148.772
C07988=1171.201,414.821,-86.704,-176.079,9.369,148.772
C07989=1171.205,414.573,-86.667,-176.079,9.367,148.771
C07990=1171.209,414.326,-86.631,-176.079,9.365,148.771
C07991=1171.213,414.079,-86.594,-176.078,9.364,148.770
C07992=1171.217,413.831,-86.558,-176.078,9.361,148.770
C07993=1171.220,413.584,-86.522,-176.078,9.360,148.769
C07994=1171.224,413.337,-86.485,-176.077,9.358,148.769
C07995=1171.228,413.089,-86.449,-176.077,9.356,148.768
C07996=1171.232,412.842,-86.413,-176.077,9.354,148.767
C07997=1171.236,412.595,-86.377,-176.077,9.353,148.767
C07998=1171.240,412.347,-86.340,-176.077,9.350,148.766
C07999=1171.244,412.100,-86.305,-176.076,9.349,148.766
C08000=1171.248,411.853,-86.268,-176.076,9.347,148.765
C08001=1171.251,411.605,-86.232,-176.076,9.345,148.765
C08002=1171.255,411.358,-86.195,-176.075,9.343,148.764
C08003=1171.259,411.110,-86.160,-176.075,9.342,148.763
C08004=1171.263,410.863,-86.123,-176.075,9.339,148.763
C08005=1171.267,410.616,-86.087,-176.074,9.338,148.762
C08006=1171.271,410.369,-86.051,-176.074,9.336,148.762
C08007=1171.275,410.121,-86.015,-176.074,9.334,148.761
C08008=1171.279,409.874,-85.978,-176.073,9.332,148.761
C08009=1171.282,409.626,-85.943,-176.073,9.329,148.760
C08010=1171.286,409.379,-85.906,-176.073,9.328,148.759
C08011=1171.291,409.131,-85.870,-176.072,9.326,148.759
C08012=1171.294,408.885,-85.833,-176.072,9.324,148.758
C08013=1171.299,408.637,-85.797,-176.072,9.322,148.758
C08014=1171.302,408.390,-85.761,-176.072,9.319,148.757
C08015=1171.306,408.142,-85.725,-176.071,9.318,148.756
C08016=1171.310,407.895,-85.689,-176.071,9.316,148.756
C08017=1171.313,407.648,-85.653,-176.071,9.314,148.755
C08018=1171.318,407.400,-85.616,-176.070,9.312,148.755
C08019=1171.321,407.153,-85.581,-176.070,9.310,148.754
C08020=1171.326,406.905,-85.544,-176.070,9.308,148.753
C08021=1171.330,406.659,-85.509,-176.070,9.306,148.753
C08022=1171.334,406.411,-85.472,-176.069,9.304,148.752
C08023=1171.337,406.164,-85.436,-176.069,9.302,148.751
C08024=1171.342,405.916,-85.400,-176.068,9.300,148.751
C08025=1171.345,405.670,-85.364,-176.068,9.297,148.750
C08026=1171.349,405.422,-85.328,-176.068,9.296,148.749
C08027=1171.353,405.175,-85.291,-176.068,9.293,148.749
C08028=1171.357,404.927,-85.255,-176.067,9.292,148.748
C08029=1171.361,404.680,-85.220,-176.067,9.289,148.748
C08030=1171.365,404.432,-85.183,-176.066,9.287,148.747
C08031=1171.369,404.185,-85.147,-176.067,9.285,148.746
C08032=1171.373,403.938,-85.110,-176.066,9.283,148.746
C08033=1171.376,403.690,-85.075,-176.066,9.281,148.745
C08034=1171.380,403.443,-85.038,-176.065,9.279,148.744
C08035=1171.384,403.196,-85.002,-176.065,9.277,148.744
C08036=1171.389,402.948,-84.966,-176.065,9.274,148.743
C08037=1171.392,402.701,-84.930,-176.064,9.272,148.743
C08038=1171.396,402.453,-84.894,-176.064,9.270,148.742
C08039=1171.400,402.206,-84.858,-176.063,9.268,148.741
C08040=1171.403,401.959,-84.822,-176.063,9.266,148.740
C08041=1171.407,401.711,-84.785,-176.064,9.263,148.740
C08042=1171.411,401.464,-84.750,-176.063,9.262,148.739
C08043=1171.416,401.217,-84.714,-176.063,9.259,148.739
C08044=1171.419,400.970,-84.678,-176.063,9.256,148.738
C08045=1171.424,400.722,-84.641,-176.062,9.255,148.737
C08046=1171.428,400.475,-84.606,-176.062,9.252,148.736
C08047=1171.432,400.227,-84.569,-176.062,9.250,148.736
C08048=1171.435,399.980,-84.533,-176.061,9.247,148.735
C08049=1171.439,399.733,-84.497,-176.061,9.246,148.735
C08050=1171.443,399.485,-84.461,-176.061,9.243,148.734
C08051=1171.447,399.238,-84.426,-176.061,9.240,148.733
C08052=1171.451,398.991,-84.389,-176.061,9.238,148.732
C08053=1171.454,398.743,-84.353,-176.060,9.236,148.732
C08054=1171.459,398.495,-84.317,-176.060,9.233,148.731
C08055=1171.462,398.248,-84.281,-176.060,9.231,148.730
C08056=1171.466,398.001,-84.245,-176.060,9.228,148.730
C08057=1171.471,397.754,-84.209,-176.059,9.226,148.729
C08058=1171.474,397.507,-84.173,-176.059,9.223,148.728
C08059=1171.479,397.259,-84.137,-176.059,9.221,148.727
C08060=1171.482,397.012,-84.101,-176.059,9.218,148.727
C08061=1171.486,396.765,-84.065,-176.058,9.216,148.726
C08062=1171.490,396.517,-84.029,-176.058,9.214,148.725
C08063=1171.494,396.269,-83.993,-176.058,9.211,148.725
C08064=1171.498,396.022,-83.957,-176.058,9.209,148.724
C08065=1171.501,395.775,-83.921,-176.058,9.206,148.723
C08066=1171.506,395.527,-83.885,-176.058,9.204,148.723
C08067=1171.509,395.280,-83.849,-176.058,9.201,148.722
C08068=1171.513,395.033,-83.813,-176.058,9.199,148.721
C08069=1171.518,394.785,-83.777,-176.057,9.196,148.721
C08070=1171.521,394.539,-83.741,-176.058,9.193,148.720
C08071=1171.525,394.291,-83.706,-176.058,9.190,148.719
C08072=1171.529,394.043,-83.669,-176.058,9.188,148.718
C08073=1171.533,393.796,-83.634,-176.057,9.185,148.718
C08074=1171.537,393.549,-83.597,-176.057,9.182,148.717
C08075=1171.541,393.301,-83.561,-176.057,9.180,148.716
C08076=1171.544,393.054,-83.526,-176.057,9.177,148.716
C08077=1171.549,392.806,-83.490,-176.057,9.174,148.715
C08078=1171.553,392.560,-83.454,-176.057,9.171,148.714
C08079=1171.556,392.312,-83.418,-176.057,9.169,148.713
C08080=1171.561,392.026,-83.377,-176.057,9.165,148.713
C08081=1171.565,391.742,-83.335,-176.057,9.163,148.712
C08082=1171.570,391.457,-83.294,-176.057,9.159,148.711
C08083=1171.575,391.172,-83.252,-176.057,9.155,148.710
C08084=1171.578,390.925,-83.217,-176.057,9.153,148.709
C08085=1171.582,390.677,-83.181,-176.058,9.150,148.709
C08086=1171.586,390.430,-83.145,-176.058,9.147,148.708
C08087=1171.590,390.183,-83.109,-176.058,9.145,148.707
C08088=1171.594,389.936,-83.074,-176.058,9.141,148.706
C08089=1171.598,389.688,-83.038,-176.058,9.139,148.706
C08090=1171.602,389.441,-83.002,-176.058,9.135,148.705
C08091=1171.606,389.193,-82.966,-176.059,9.132,148.704
C08092=1171.609,388.946,-82.930,-176.059,9.129,148.703
C08093=1171.613,388.698,-82.894,-176.059,9.126,148.703
C08094=1171.617,388.451,-82.859,-176.059,9.124,148.702
C08095=1171.621,388.204,-82.823,-176.060,9.120,148.701
C08096=1171.626,387.956,-82.787,-176.060,9.117,148.701
C08097=1171.629,387.709,-82.752,-176.060,9.114,148.700
C08098=1171.633,387.462,-82.715,-176.060,9.111,148.699
C08099=1171.636,387.214,-82.680,-176.061,9.108,148.699
C08100=1171.641,386.967,-82.644,-176.061,9.105,148.698
C08101=1171.645,386.720,-82.609,-176.061,9.102,148.697
C08102=1171.649,386.472,-82.573,-176.062,9.098,148.696
C08103=1171.653,386.225,-82.537,-176.063,9.095,148.696
C08104=1171.657,385.977,-82.501,-176.063,9.092,148.695
C08105=1171.661,385.730,-82.466,-176.063,9.089,148.694
C08106=1171.664,385.482,-82.430,-176.064,9.086,148.694
C08107=1171.669,385.235,-82.394,-176.064,9.083,148.693
C08108=1171.673,384.987,-82.359,-176.065,9.080,148.692
C08109=1171.676,384.741,-82.323,-176.065,9.076,148.691
C08110=1171.680,384.493,-82.287,-176.066,9.073,148.691
C08111=1171.684,384.246,-82.252,-176.067,9.070,148.690
C08112=1171.688,383.998,-82.215,-176.068,9.066,148.689
C08113=1171.692,383.751,-82.180,-176.069,9.063,148.689
C08114=1171.696,383.503,-82.145,-176.069,9.059,148.688
C08115=1171.700,383.256,-82.109,-176.070,9.056,148.687
C08116=1171.704,383.008,-82.073,-176.070,9.053,148.687
C08117=1171.708,382.761,-82.037,-176.071,9.050,148.686
C08118=1171.712,382.514,-82.002,-176.071,9.046,148.685
C08119=1171.716,382.266,-81.967,-176.073,9.042,148.685
C08120=1171.719,382.019,-81.931,-176.073,9.039,148.684
C08121=1171.723,381.771,-81.896,-176.074,9.036,148.683
C08122=1171.728,381.524,-81.861,-176.075,9.033,148.683
C08123=1171.732,381.276,-81.825,-176.076,9.029,148.682
C08124=1171.735,381.029,-81.789,-176.077,9.026,148.681
C08125=1171.739,380.781,-81.754,-176.078,9.022,148.681
C08126=1171.743,380.534,-81.718,-176.079,9.019,148.680
C08127=1171.747,380.287,-81.683,-176.079,9.015,148.679
C08128=1171.751,380.039,-81.647,-176.080,9.012,148.679
C08129=1171.755,379.791,-81.611,-176.082,9.008,148.678
C08130=1171.759,379.544,-81.576,-176.083,9.005,148.678
C08131=1171.763,379.297,-81.541,-176.084,9.001,148.677
C08132=1171.767,379.049,-81.506,-176.084,8.998,148.676
C08133=1171.771,378.802,-81.470,-176.086,8.994,148.675
C08134=1171.774,378.554,-81.435,-176.087,8.991,148.675
C08135=1171.779,378.307,-81.400,-176.088,8.987,148.674
C08136=1171.783,378.059,-81.363,-176.089,8.984,148.674
C08137=1171.787,377.811,-81.329,-176.090,8.980,148.673
C08138=1171.791,377.565,-81.293,-176.091,8.977,148.673
C08139=1171.795,377.317,-81.258,-176.093,8.973,148.672
C08140=1171.799,377.070,-81.222,-176.094,8.969,148.671
C08141=1171.802,376.822,-81.187,-176.095,8.966,148.671
C08142=1171.807,376.575,-81.152,-176.096,8.962,148.670
C08143=1171.810,376.327,-81.117,-176.097,8.959,148.670
C08144=1171.814,376.080,-81.081,-176.099,8.955,148.669
C08145=1171.818,375.833,-81.046,-176.100,8.951,148.668
C08146=1171.822,375.585,-81.011,-176.102,8.947,148.668
C08147=1171.826,375.337,-80.976,-176.103,8.944,148.667
C08148=1171.830,375.090,-80.940,-176.104,8.941,148.667
C08149=1171.834,374.842,-80.906,-176.106,8.937,148.666
C08150=1171.838,374.595,-80.870,-176.107,8.933,148.666
C08151=1171.842,374.347,-80.835,-176.108,8.930,148.665
C08152=1171.846,374.100,-80.800,-176.110,8.926,148.665
C08153=1171.850,373.852,-80.765,-176.111,8.922,148.664
C08154=1171.853,373.605,-80.729,-176.113,8.919,148.663
C08155=1171.858,373.357,-80.695,-176.115,8.915,148.663
C08156=1171.862,373.110,-80.659,-176.115,8.912,148.662
C08157=1171.866,372.863,-80.625,-176.117,8.908,148.662
C08158=1171.870,372.615,-80.589,-176.119,8.904,148.661
C08159=1171.874,372.367,-80.554,-176.120,8.901,148.661
C08160=1171.878,372.120,-80.519,-176.122,8.897,148.660
C08161=1171.882,371.873,-80.483,-176.124,8.893,148.660
C08162=1171.885,371.625,-80.449,-176.126,8.889,148.659
C08163=1171.889,371.378,-80.414,-176.127,8.885,148.659
C08164=1171.893,371.130,-80.379,-176.129,8.882,148.658
C08165=1171.897,370.882,-80.344,-176.130,8.878,148.658
C08166=1171.902,370.635,-80.309,-176.132,8.874,148.657
C08167=1171.905,370.387,-80.274,-176.134,8.871,148.657
C08168=1171.910,370.140,-80.239,-176.136,8.867,148.656
C08169=1171.914,369.892,-80.204,-176.137,8.863,148.656
C08170=1171.917,369.644,-80.169,-176.139,8.860,148.655
C08171=1171.921,369.397,-80.135,-176.141,8.856,148.655
C08172=1171.925,369.150,-80.099,-176.143,8.852,148.654
C08173=1171.929,368.902,-80.065,-176.145,8.849,148.654
C08174=1171.933,368.654,-80.030,-176.146,8.845,148.653
C08175=1171.938,368.407,-79.995,-176.148,8.841,148.653
C08176=1171.941,368.160,-79.961,-176.150,8.838,148.652
C08177=1171.945,367.912,-79.925,-176.151,8.834,148.652
C08178=1171.949,367.665,-79.891,-176.153,8.830,148.652
C08179=1171.953,367.417,-79.856,-176.155,8.827,148.651
C08180=1171.958,367.169,-79.821,-176.158,8.822,148.651
C08181=1171.961,366.922,-79.786,-176.159,8.819,148.650
C08182=1171.965,366.675,-79.752,-176.161,8.815,148.650
C08183=1171.969,366.426,-79.717,-176.163,8.812,148.649
C08184=1171.974,366.145,-79.678,-176.166,8.807,148.649
C08185=1171.978,365.862,-79.638,-176.167,8.804,148.649
C08186=1171.983,365.581,-79.598,-176.170,8.799,148.648
C08187=1171.987,365.298,-79.559,-176.172,8.795,148.648
C08188=1171.991,365.051,-79.525,-176.174,8.791,148.647
C08189=1171.995,364.803,-79.490,-176.176,8.788,148.647
C08190=1172.000,364.556,-79.455,-176.178,8.784,148.646
C08191=1172.003,364.309,-79.420,-176.181,8.780,148.646
C08192=1172.007,364.061,-79.386,-176.182,8.776,148.646
C08193=1172.011,363.813,-79.351,-176.185,8.773,148.645
C08194=1172.015,363.566,-79.317,-176.187,8.769,148.645
C08195=1172.019,363.318,-79.282,-176.188,8.766,148.644
C08196=1172.023,363.071,-79.249,-176.191,8.761,148.644
C08197=1172.027,362.823,-79.214,-176.193,8.758,148.644
C08198=1172.031,362.575,-79.179,-176.195,8.754,148.643
C08199=1172.035,362.327,-79.145,-176.197,8.751,148.643
C08200=1172.039,362.080,-79.111,-176.200,8.747,148.643
C08201=1172.043,361.832,-79.076,-176.201,8.743,148.642
C08202=1172.047,361.585,-79.041,-176.204,8.740,148.642
C08203=1172.051,361.338,-79.007,-176.206,8.736,148.642
C08204=1172.055,361.090,-78.972,-176.208,8.732,148.641
C08205=1172.059,360.842,-78.939,-176.210,8.728,148.641
C08206=1172.063,360.594,-78.904,-176.213,8.725,148.641
C08207=1172.067,360.347,-78.870,-176.214,8.721,148.640
C08208=1172.070,360.099,-78.836,-176.217,8.717,148.640
C08209=1172.075,359.852,-78.801,-176.219,8.714,148.640
C08210=1172.080,359.604,-78.767,-176.221,8.710,148.639
C08211=1172.083,359.356,-78.733,-176.224,8.707,148.639
C08212=1172.087,359.109,-78.698,-176.226,8.703,148.639
C08213=1172.091,358.861,-78.664,-176.228,8.699,148.638
C08214=1172.095,358.614,-78.629,-176.230,8.696,148.638
C08215=1172.099,358.366,-78.596,-176.232,8.692,148.638
C08216=1172.103,358.118,-78.562,-176.235,8.688,148.637
C08217=1172.107,357.871,-78.527,-176.237,8.685,148.637
C08218=1172.111,357.624,-78.494,-176.239,8.681,148.637
C08219=1172.115,357.376,-78.459,-176.242,8.678,148.637
C08220=1172.119,357.128,-78.426,-176.244,8.674,148.636
C08221=1172.124,356.880,-78.391,-176.246,8.670,148.636
C08222=1172.127,356.633,-78.357,-176.249,8.667,148.636
C08223=1172.131,356.385,-78.322,-176.251,8.663,148.635
C08224=1172.136,356.137,-78.289,-176.253,8.659,148.635
C08225=1172.139,355.890,-78.255,-176.256,8.656,148.635
C08226=1172.143,355.642,-78.221,-176.258,8.652,148.634
C08227=1172.148,355.395,-78.187,-176.260,8.648,148.634
C08228=1172.152,355.146,-78.153,-176.263,8.645,148.634
C08229=1172.155,354.899,-78.119,-176.265,8.642,148.634
C08230=1172.159,354.652,-78.086,-176.267,8.638,148.633
C08231=1172.163,354.403,-78.051,-176.269,8.635,148.633
C08232=1172.167,354.156,-78.017,-176.272,8.631,148.633
C08233=1172.171,353.909,-77.984,-176.274,8.627,148.633
C08234=1172.176,353.661,-77.949,-176.276,8.624,148.632
C08235=1172.180,353.413,-77.916,-176.278,8.620,148.632
C08236=1172.183,353.166,-77.882,-176.281,8.616,148.632
C08237=1172.188,352.918,-77.848,-176.283,8.613,148.631
C08238=1172.191,352.670,-77.814,-176.286,8.610,148.631
C08239=1172.196,352.422,-77.781,-176.288,8.606,148.631
C08240=1172.199,352.175,-77.747,-176.290,8.602,148.630
C08241=1172.204,351.927,-77.713,-176.293,8.599,148.630
C08242=1172.208,351.680,-77.679,-176.295,8.595,148.630
C08243=1172.212,351.431,-77.646,-176.297,8.592,148.630
C08244=1172.216,351.184,-77.612,-176.300,8.589,148.630
C08245=1172.220,350.936,-77.578,-176.302,8.584,148.629
C08246=1172.224,350.689,-77.544,-176.304,8.581,148.629
C08247=1172.228,350.441,-77.511,-176.306,8.578,148.629
C08248=1172.232,350.193,-77.478,-176.309,8.574,148.628
C08249=1172.236,349.946,-77.443,-176.312,8.570,148.628
C08250=1172.241,349.698,-77.410,-176.314,8.567,148.628
C08251=1172.244,349.451,-77.376,-176.316,8.564,148.628
C08252=1172.248,349.202,-77.343,-176.318,8.560,148.628
C08253=1172.252,348.955,-77.309,-176.321,8.557,148.627
C08254=1172.256,348.707,-77.276,-176.323,8.553,148.627
C08255=1172.261,348.459,-77.242,-176.325,8.549,148.627
C08256=1172.265,348.212,-77.209,-176.328,8.546,148.626
C08257=1172.269,347.964,-77.175,-176.330,8.543,148.626
C08258=1172.273,347.717,-77.142,-176.332,8.539,148.626
C08259=1172.276,347.468,-77.108,-176.335,8.535,148.626
C08260=1172.281,347.221,-77.075,-176.337,8.532,148.626
C08261=1172.285,346.973,-77.042,-176.340,8.529,148.625
C08262=1172.289,346.725,-77.009,-176.342,8.525,148.625
C08263=1172.293,346.478,-76.974,-176.344,8.522,148.625
C08264=1172.298,346.230,-76.941,-176.347,8.518,148.625
C08265=1172.302,345.982,-76.908,-176.349,8.515,148.624
C08266=1172.306,345.735,-76.875,-176.352,8.511,148.624
C08267=1172.309,345.486,-76.841,-176.354,8.508,148.624
C08268=1172.314,345.238,-76.808,-176.356,8.505,148.624
C08269=1172.318,344.991,-76.775,-176.358,8.501,148.624
C08270=1172.322,344.743,-76.742,-176.361,8.497,148.623
C08271=1172.326,344.496,-76.708,-176.364,8.494,148.623
C08272=1172.330,344.248,-76.675,-176.366,8.491,148.623
C08273=1172.334,344.000,-76.641,-176.368,8.487,148.623
C08274=1172.338,343.753,-76.608,-176.370,8.484,148.622
C08275=1172.342,343.505,-76.575,-176.373,8.481,148.622
C08276=1172.346,343.257,-76.542,-176.376,8.477,148.622
C08277=1172.350,343.010,-76.509,-176.378,8.473,148.622
C08278=1172.355,342.762,-76.476,-176.380,8.470,148.622
C08279=1172.359,342.514,-76.443,-176.382,8.467,148.621
C08280=1172.363,342.266,-76.409,-176.385,8.463,148.621
C08281=1172.367,342.018,-76.377,-176.387,8.460,148.621
C08282=1172.371,341.770,-76.344,-176.390,8.456,148.621
C08283=1172.376,341.523,-76.311,-176.393,8.453,148.621
C08284=1172.380,341.275,-76.277,-176.395,8.450,148.620
C08285=1172.384,341.027,-76.244,-176.397,8.446,148.620
C08286=1172.387,340.780,-76.212,-176.399,8.443,148.620
C08287=1172.391,340.532,-76.179,-176.402,8.440,148.620
C08288=1172.396,340.252,-76.141,-176.405,8.436,148.620
C08289=1172.401,339.973,-76.104,-176.407,8.432,148.619
C08290=1172.405,339.694,-76.068,-176.410,8.429,148.619
C08291=1172.410,339.414,-76.030,-176.413,8.424,148.619
C08292=1172.414,339.166,-75.997,-176.415,8.421,148.619
C08293=1172.418,338.919,-75.964,-176.418,8.418,148.619
C08294=1172.422,338.671,-75.931,-176.420,8.414,148.618
C08295=1172.426,338.423,-75.899,-176.423,8.410,148.618
C08296=1172.430,338.175,-75.866,-176.425,8.407,148.618
C08297=1172.434,337.927,-75.833,-176.428,8.404,148.618
C08298=1172.439,337.679,-75.800,-176.430,8.401,148.618
C08299=1172.443,337.431,-75.767,-176.432,8.398,148.618
C08300=1172.446,337.184,-75.734,-176.434,8.394,148.617
C08301=1172.451,336.937,-75.702,-176.437,8.391,148.617
C08302=1172.456,336.688,-75.669,-176.440,8.387,148.617
C08303=1172.459,336.441,-75.637,-176.442,8.384,148.617
C08304=1172.463,336.193,-75.604,-176.445,8.381,148.617
C08305=1172.468,335.945,-75.571,-176.447,8.377,148.616
C08306=1172.472,335.697,-75.538,-176.449,8.374,148.616
C08307=1172.475,335.449,-75.506,-176.452,8.371,148.616
C08308=1172.480,335.201,-75.473,-176.454,8.368,148.616
C08309=1172.484,334.953,-75.440,-176.456,8.364,148.616
C08310=1172.487,334.706,-75.408,-176.459,8.360,148.616
C08311=1172.492,334.457,-75.375,-176.462,8.357,148.616
C08312=1172.497,334.210,-75.343,-176.464,8.354,148.615
C08313=1172.500,333.962,-75.311,-176.467,8.351,148.615
C08314=1172.504,333.715,-75.278,-176.469,8.347,148.615
C08315=1172.509,333.466,-75.245,-176.472,8.344,148.615
C08316=1172.512,333.219,-75.213,-176.474,8.341,148.615
C08317=1172.517,332.970,-75.180,-176.476,8.338,148.615
C08318=1172.521,332.723,-75.147,-176.479,8.334,148.614
C08319=1172.525,332.475,-75.116,-176.482,8.331,148.614
C08320=1172.530,332.227,-75.083,-176.484,8.327,148.614
C08321=1172.533,331.980,-75.051,-176.486,8.324,148.614
C08322=1172.537,331.731,-75.018,-176.489,8.321,148.614
C08323=1172.541,331.484,-74.986,-176.491,8.318,148.614
C08324=1172.546,331.236,-74.953,-176.494,8.314,148.613
C08325=1172.550,330.988,-74.921,-176.496,8.311,148.613
C08326=1172.554,330.740,-74.888,-176.499,8.308,148.613
C08327=1172.558,330.492,-74.856,-176.501,8.305,148.613
C08328=1172.562,330.244,-74.824,-176.504,8.301,148.613
C08329=1172.567,329.996,-74.792,-176.506,8.298,148.613
C08330=1172.570,329.749,-74.760,-176.509,8.294,148.613
C08331=1172.575,329.501,-74.727,-176.511,8.291,148.612
C08332=1172.578,329.253,-74.695,-176.514,8.288,148.612
C08333=1172.583,329.005,-74.663,-176.516,8.285,148.612
C08334=1172.587,328.757,-74.631,-176.518,8.282,148.612
C08335=1172.591,328.509,-74.598,-176.521,8.279,148.612
C08336=1172.595,328.261,-74.566,-176.523,8.275,148.612
C08337=1172.600,328.013,-74.534,-176.526,8.272,148.612
C08338=1172.604,327.765,-74.502,-176.528,8.269,148.612
C08339=1172.607,327.518,-74.470,-176.531,8.265,148.611
C08340=1172.612,327.270,-74.437,-176.533,8.261,148.611
C08341=1172.616,327.022,-74.406,-176.536,8.259,148.611
C08342=1172.620,326.774,-74.373,-176.538,8.255,148.611
C08343=1172.624,326.526,-74.342,-176.541,8.252,148.611
C08344=1172.628,326.278,-74.310,-176.543,8.249,148.611
C08345=1172.633,326.030,-74.278,-176.546,8.246,148.611
C08346=1172.637,325.782,-74.246,-176.548,8.243,148.611
C08347=1172.641,325.534,-74.213,-176.551,8.239,148.610
C08348=1172.645,325.286,-74.182,-176.553,8.236,148.610
C08349=1172.649,325.038,-74.150,-176.556,8.233,148.610
C08350=1172.653,324.790,-74.118,-176.558,8.230,148.610
C08351=1172.658,324.543,-74.086,-176.561,8.227,148.610
C08352=1172.661,324.295,-74.054,-176.563,8.223,148.610
C08353=1172.666,324.046,-74.022,-176.566,8.219,148.610
C08354=1172.670,323.799,-73.990,-176.569,8.216,148.610
C08355=1172.674,323.551,-73.959,-176.571,8.213,148.609
C08356=1172.678,323.303,-73.927,-176.574,8.210,148.609
C08357=1172.683,323.055,-73.895,-176.576,8.207,148.609
C08358=1172.686,322.807,-73.863,-176.578,8.203,148.609
C08359=1172.690,322.559,-73.831,-176.581,8.200,148.609
C08360=1172.695,322.311,-73.800,-176.583,8.197,148.609
C08361=1172.699,322.063,-73.768,-176.586,8.194,148.609
C08362=1172.703,321.815,-73.736,-176.588,8.191,148.609
C08363=1172.707,321.568,-73.704,-176.591,8.188,148.609
C08364=1172.711,321.319,-73.673,-176.593,8.185,148.608
C08365=1172.715,321.072,-73.641,-176.596,8.182,148.608
C08366=1172.720,320.823,-73.609,-176.598,8.178,148.608
C08367=1172.724,320.575,-73.578,-176.601,8.175,148.608
C08368=1172.728,320.328,-73.546,-176.603,8.172,148.608
C08369=1172.732,320.080,-73.514,-176.605,8.169,148.608
C08370=1172.736,319.832,-73.483,-176.608,8.166,148.608
C08371=1172.741,319.583,-73.451,-176.611,8.162,148.608
C08372=1172.744,319.335,-73.419,-176.614,8.159,148.608
C08373=1172.749,319.087,-73.388,-176.616,8.155,148.607
C08374=1172.753,318.839,-73.357,-176.619,8.152,148.607
C08375=1172.757,318.592,-73.325,-176.621,8.149,148.607
C08376=1172.761,318.343,-73.294,-176.624,8.146,148.607
C08377=1172.765,318.096,-73.262,-176.626,8.143,148.607
C08378=1172.769,317.848,-73.231,-176.629,8.140,148.607
C08379=1172.774,317.600,-73.200,-176.631,8.136,148.607
C08380=1172.778,317.352,-73.167,-176.634,8.133,148.607
C08381=1172.782,317.104,-73.136,-176.636,8.130,148.607
C08382=1172.786,316.856,-73.105,-176.639,8.127,148.607
C08383=1172.791,316.608,-73.073,-176.641,8.124,148.606
C08384=1172.795,316.360,-73.042,-176.644,8.121,148.606
C08385=1172.799,316.112,-73.011,-176.646,8.118,148.606
C08386=1172.803,315.864,-72.980,-176.649,8.115,148.606
C08387=1172.807,315.616,-72.948,-176.651,8.111,148.606
C08388=1172.811,315.368,-72.917,-176.654,8.108,148.606
C08389=1172.816,315.120,-72.885,-176.657,8.105,148.606
C08390=1172.820,314.872,-72.854,-176.659,8.102,148.606
C08391=1172.824,314.624,-72.823,-176.662,8.099,148.606
C08392=1172.829,314.347,-72.789,-176.664,8.095,148.606
C08393=1172.833,314.070,-72.754,-176.667,8.092,148.606
C08394=1172.838,313.794,-72.718,-176.670,8.088,148.605
C08395=1172.842,313.516,-72.683,-176.673,8.085,148.605
C08396=1172.847,313.269,-72.653,-176.676,8.082,148.605
C08397=1172.851,313.021,-72.622,-176.678,8.079,148.605
C08398=1172.855,312.773,-72.590,-176.681,8.076,148.605
C08399=1172.859,312.525,-72.559,-176.683,8.072,148.605
C08400=1172.863,312.276,-72.528,-176.686,8.069,148.605
C08401=1172.868,312.029,-72.497,-176.688,8.066,148.605
C08402=1172.872,311.781,-72.466,-176.691,8.063,148.605
C08403=1172.876,311.532,-72.435,-176.693,8.060,148.605
C08404=1172.880,311.284,-72.405,-176.696,8.057,148.605
C08405=1172.884,311.036,-72.373,-176.698,8.054,148.605
C08406=1172.889,310.788,-72.342,-176.701,8.050,148.605
C08407=1172.893,310.540,-72.311,-176.703,8.047,148.605
C08408=1172.897,310.292,-72.280,-176.706,8.044,148.605
C08409=1172.902,310.044,-72.249,-176.708,8.041,148.604
C08410=1172.906,309.796,-72.218,-176.711,8.038,148.604
C08411=1172.909,309.548,-72.187,-176.713,8.035,148.604
C08412=1172.914,309.300,-72.157,-176.716,8.032,148.604
C08413=1172.918,309.051,-72.125,-176.719,8.029,148.604
C08414=1172.923,308.803,-72.095,-176.721,8.026,148.604
C08415=1172.927,308.555,-72.064,-176.724,8.023,148.604
C08416=1172.931,308.307,-72.033,-176.726,8.019,148.604
C08417=1172.935,308.060,-72.002,-176.729,8.016,148.604
C08418=1172.939,307.812,-71.971,-176.732,8.013,148.604
C08419=1172.943,307.563,-71.940,-176.734,8.010,148.604
C08420=1172.947,307.316,-71.910,-176.737,8.007,148.604
C08421=1172.952,307.068,-71.879,-176.739,8.004,148.604
C08422=1172.957,306.820,-71.848,-176.742,8.001,148.604
C08423=1172.961,306.571,-71.817,-176.744,7.998,148.604
C08424=1172.964,306.323,-71.787,-176.747,7.995,148.603
C08425=1172.969,306.075,-71.756,-176.749,7.992,148.603
C08426=1172.973,305.827,-71.725,-176.752,7.989,148.604
C08427=1172.977,305.579,-71.695,-176.754,7.985,148.603
C08428=1172.982,305.331,-71.664,-176.757,7.982,148.603
C08429=1172.986,305.083,-71.633,-176.760,7.979,148.603
C08430=1172.990,304.834,-71.604,-176.762,7.976,148.603
C08431=1172.994,304.586,-71.573,-176.765,7.973,148.603
C08432=1172.999,304.338,-71.542,-176.768,7.970,148.603
C08433=1173.003,304.091,-71.512,-176.770,7.967,148.603
C08434=1173.007,303.842,-71.481,-176.773,7.964,148.603
C08435=1173.012,303.594,-71.450,-176.775,7.961,148.603
C08436=1173.015,303.346,-71.420,-176.777,7.958,148.603
C08437=1173.020,303.098,-71.389,-176.780,7.955,148.603
C08438=1173.024,302.849,-71.359,-176.782,7.952,148.603
C08439=1173.028,302.601,-71.329,-176.785,7.949,148.603
C08440=1173.033,302.354,-71.298,-176.787,7.946,148.603
C08441=1173.037,302.106,-71.268,-176.790,7.943,148.603
C08442=1173.042,301.857,-71.238,-176.792,7.940,148.603
C08443=1173.045,301.609,-71.207,-176.795,7.937,148.603
C08444=1173.050,301.361,-71.176,-176.798,7.934,148.603
C08445=1173.053,301.113,-71.146,-176.800,7.931,148.603
C08446=1173.058,300.865,-71.116,-176.803,7.928,148.603
C08447=1173.062,300.617,-71.086,-176.806,7.925,148.603
C08448=1173.067,300.369,-71.055,-176.808,7.922,148.603
C08449=1173.070,300.120,-71.025,-176.811,7.918,148.602
C08450=1173.075,299.872,-70.995,-176.813,7.915,148.602
C08451=1173.079,299.625,-70.964,-176.816,7.912,148.602
C08452=1173.084,299.376,-70.934,-176.818,7.909,148.602
C08453=1173.088,299.128,-70.904,-176.821,7.906,148.602
C08454=1173.093,298.880,-70.874,-176.824,7.903,148.602
C08455=1173.096,298.632,-70.844,-176.827,7.900,148.602
C08456=1173.100,298.383,-70.813,-176.828,7.898,148.602
C08457=1173.105,298.135,-70.783,-176.831,7.895,148.602
C08458=1173.109,297.888,-70.753,-176.834,7.892,148.602
C08459=1173.113,297.639,-70.723,-176.836,7.888,148.602
C08460=1173.117,297.391,-70.693,-176.839,7.885,148.602
C08461=1173.122,297.143,-70.663,-176.842,7.882,148.602
C08462=1173.126,296.895,-70.633,-176.844,7.879,148.602
C08463=1173.130,296.647,-70.603,-176.847,7.876,148.602
C08464=1173.135,296.399,-70.573,-176.849,7.873,148.602
C08465=1173.138,296.150,-70.543,-176.852,7.870,148.602
C08466=1173.142,295.902,-70.513,-176.855,7.867,148.602
C08467=1173.147,295.654,-70.482,-176.857,7.864,148.602
C08468=1173.151,295.405,-70.453,-176.860,7.861,148.602
C08469=1173.155,295.158,-70.423,-176.862,7.859,148.602
C08470=1173.160,294.909,-70.393,-176.865,7.856,148.602
C08471=1173.164,294.662,-70.363,-176.867,7.852,148.602
C08472=1173.168,294.413,-70.333,-176.870,7.849,148.602
C08473=1173.173,294.165,-70.303,-176.872,7.846,148.602
C08474=1173.177,293.917,-70.273,-176.875,7.844,148.602
C08475=1173.181,293.669,-70.244,-176.878,7.841,148.602
C08476=1173.185,293.421,-70.214,-176.880,7.837,148.602
C08477=1173.190,293.173,-70.183,-176.883,7.834,148.602
C08478=1173.194,292.924,-70.154,-176.886,7.831,148.602
C08479=1173.198,292.676,-70.124,-176.888,7.828,148.602
C08480=1173.203,292.428,-70.095,-176.891,7.825,148.602
C08481=1173.207,292.180,-70.064,-176.893,7.823,148.602
C08482=1173.211,291.932,-70.035,-176.896,7.820,148.602
C08483=1173.216,291.683,-70.005,-176.898,7.817,148.602
C08484=1173.220,291.435,-69.976,-176.901,7.814,148.602
C08485=1173.224,291.187,-69.946,-176.903,7.811,148.602
C08486=1173.228,290.939,-69.916,-176.906,7.808,148.602
C08487=1173.233,290.690,-69.886,-176.909,7.805,148.602
C08488=1173.237,290.442,-69.857,-176.912,7.802,148.602
C08489=1173.241,290.194,-69.827,-176.914,7.799,148.602
C08490=1173.245,289.946,-69.798,-176.917,7.795,148.602
C08491=1173.249,289.697,-69.768,-176.919,7.793,148.602
C08492=1173.254,289.449,-69.739,-176.922,7.790,148.602
C08493=1173.258,289.201,-69.709,-176.924,7.787,148.602
C08494=1173.262,288.953,-69.679,-176.927,7.784,148.602
C08495=1173.267,288.705,-69.649,-176.930,7.781,148.602
C08496=1173.271,288.430,-69.618,-176.932,7.778,148.602
C08497=1173.276,288.156,-69.584,-176.935,7.774,148.602
C08498=1173.281,287.880,-69.552,-176.938,7.771,148.602
C08499=1173.285,287.605,-69.520,-176.941,7.768,148.602
C08500=1173.290,287.357,-69.490,-176.944,7.765,148.602
C08501=1173.295,287.109,-69.461,-176.946,7.762,148.602
C08502=1173.299,286.861,-69.431,-176.949,7.759,148.602
C08503=1173.303,286.612,-69.402,-176.952,7.756,148.602
C08504=1173.307,286.364,-69.372,-176.954,7.753,148.602
C08505=1173.312,286.116,-69.343,-176.956,7.751,148.602
C08506=1173.316,285.868,-69.313,-176.959,7.748,148.602
C08507=1173.320,285.619,-69.284,-176.962,7.745,148.602
C08508=1173.324,285.371,-69.254,-176.964,7.742,148.602
C08509=1173.329,285.124,-69.225,-176.967,7.739,148.602
C08510=1173.333,284.875,-69.196,-176.970,7.736,148.602
C08511=1173.338,284.626,-69.167,-176.972,7.733,148.602
C08512=1173.342,284.378,-69.138,-176.974,7.731,148.602
C08513=1173.346,284.130,-69.108,-176.977,7.728,148.602
C08514=1173.349,283.882,-69.079,-176.980,7.725,148.602
C08515=1173.354,283.634,-69.050,-176.983,7.722,148.602
C08516=1173.359,283.385,-69.021,-176.985,7.719,148.602
C08517=1173.363,283.137,-68.992,-176.988,7.716,148.602
C08518=1173.367,282.889,-68.963,-176.991,7.713,148.602
C08519=1173.371,282.641,-68.933,-176.992,7.710,148.602
C08520=1173.376,282.392,-68.905,-176.995,7.707,148.602
C08521=1173.381,282.144,-68.875,-176.998,7.704,148.602
C08522=1173.385,281.896,-68.846,-177.001,7.701,148.602
C08523=1173.389,281.647,-68.817,-177.003,7.698,148.602
C08524=1173.393,281.399,-68.788,-177.006,7.695,148.602
C08525=1173.397,281.151,-68.759,-177.009,7.692,148.602
C08526=1173.402,280.903,-68.730,-177.011,7.690,148.602
C08527=1173.406,280.654,-68.701,-177.014,7.687,148.602
C08528=1173.410,280.406,-68.671,-177.017,7.684,148.602
C08529=1173.415,280.158,-68.643,-177.019,7.681,148.602
C08530=1173.419,279.910,-68.614,-177.022,7.678,148.602
C08531=1173.423,279.661,-68.586,-177.024,7.675,148.602
C08532=1173.427,279.413,-68.556,-177.026,7.673,148.602
C08533=1173.432,279.165,-68.527,-177.029,7.670,148.602
C08534=1173.436,278.917,-68.499,-177.032,7.667,148.602
C08535=1173.440,278.668,-68.469,-177.035,7.664,148.602
C08536=1173.445,278.419,-68.441,-177.037,7.661,148.602
C08537=1173.449,278.172,-68.412,-177.040,7.658,148.603
C08538=1173.453,277.923,-68.383,-177.042,7.656,148.603
C08539=1173.457,277.675,-68.354,-177.045,7.653,148.603
C08540=1173.462,277.427,-68.326,-177.048,7.650,148.603
C08541=1173.467,277.179,-68.296,-177.051,7.647,148.603
C08542=1173.470,276.930,-68.268,-177.053,7.644,148.603
C08543=1173.476,276.682,-68.240,-177.055,7.642,148.603
C08544=1173.480,276.434,-68.210,-177.058,7.639,148.603
C08545=1173.483,276.185,-68.182,-177.061,7.636,148.603
C08546=1173.488,275.937,-68.153,-177.063,7.633,148.603
C08547=1173.493,275.689,-68.124,-177.066,7.630,148.603
C08548=1173.496,275.440,-68.096,-177.069,7.627,148.603
C08549=1173.501,275.192,-68.067,-177.071,7.625,148.603
C08550=1173.506,274.943,-68.038,-177.074,7.622,148.603
C08551=1173.509,274.695,-68.010,-177.076,7.619,148.603
C08552=1173.514,274.447,-67.981,-177.079,7.616,148.603
C08553=1173.518,274.199,-67.953,-177.082,7.613,148.603
C08554=1173.523,273.950,-67.924,-177.084,7.610,148.603
C08555=1173.528,273.702,-67.896,-177.087,7.607,148.603
C08556=1173.531,273.454,-67.867,-177.090,7.605,148.603
C08557=1173.536,273.206,-67.839,-177.092,7.602,148.603
C08558=1173.540,272.957,-67.810,-177.095,7.599,148.603
C08559=1173.544,272.708,-67.782,-177.097,7.596,148.603
C08560=1173.548,272.461,-67.753,-177.100,7.593,148.603
C08561=1173.553,272.212,-67.724,-177.103,7.590,148.604
C08562=1173.558,271.964,-67.696,-177.105,7.588,148.604
C08563=1173.562,271.715,-67.668,-177.108,7.585,148.604
C08564=1173.566,271.466,-67.639,-177.110,7.582,148.604
C08565=1173.571,271.218,-67.611,-177.113,7.579,148.604
C08566=1173.575,270.970,-67.582,-177.116,7.576,148.604
C08567=1173.579,270.722,-67.554,-177.119,7.573,148.604
C08568=1173.584,270.473,-67.525,-177.121,7.571,148.604
C08569=1173.588,270.226,-67.498,-177.123,7.568,148.604
C08570=1173.592,269.977,-67.469,-177.126,7.565,148.604
C08571=1173.597,269.729,-67.441,-177.129,7.562,148.604
C08572=1173.601,269.480,-67.413,-177.131,7.560,148.604
C08573=1173.605,269.231,-67.384,-177.134,7.557,148.604
C08574=1173.609,268.983,-67.356,-177.137,7.554,148.604
C08575=1173.614,268.735,-67.328,-177.139,7.551,148.604
C08576=1173.618,268.487,-67.300,-177.142,7.548,148.604
C08577=1173.623,268.238,-67.271,-177.144,7.546,148.604
C08578=1173.627,267.990,-67.243,-177.147,7.543,148.605
C08579=1173.631,267.741,-67.215,-177.150,7.540,148.605
C08580=1173.636,267.493,-67.187,-177.153,7.537,148.605
C08581=1173.640,267.245,-67.159,-177.155,7.535,148.605
C08582=1173.644,266.997,-67.131,-177.157,7.532,148.605
C08583=1173.649,266.749,-67.103,-177.160,7.529,148.605
C08584=1173.653,266.500,-67.074,-177.163,7.527,148.605
C08585=1173.658,266.251,-67.047,-177.166,7.524,148.605
C08586=1173.662,266.003,-67.019,-177.168,7.521,148.605
C08587=1173.666,265.755,-66.991,-177.171,7.518,148.605
C08588=1173.671,265.506,-66.962,-177.174,7.516,148.605
C08589=1173.675,265.258,-66.934,-177.176,7.513,148.605
C08590=1173.679,265.009,-66.906,-177.179,7.510,148.605
C08591=1173.684,264.761,-66.879,-177.181,7.507,148.605
C08592=1173.689,264.513,-66.851,-177.184,7.504,148.606
C08593=1173.692,264.264,-66.823,-177.186,7.502,148.606
C08594=1173.697,264.016,-66.795,-177.189,7.499,148.606
C08595=1173.702,263.767,-66.767,-177.192,7.496,148.606
C08596=1173.706,263.519,-66.739,-177.195,7.493,148.606
C08597=1173.710,263.270,-66.711,-177.197,7.491,148.606
C08598=1173.714,263.022,-66.683,-177.200,7.488,148.606
C08599=1173.719,262.774,-66.656,-177.203,7.486,148.606
C08600=1173.723,262.501,-66.625,-177.205,7.483,148.606
C08601=1173.728,262.227,-66.595,-177.208,7.480,148.606
C08602=1173.733,261.955,-66.564,-177.211,7.477,148.606
C08603=1173.738,261.682,-66.533,-177.214,7.474,148.606
C08604=1173.742,261.433,-66.506,-177.217,7.471,148.607
C08605=1173.747,261.184,-66.477,-177.220,7.468,148.607
C08606=1173.751,260.936,-66.450,-177.222,7.466,148.607
C08607=1173.756,260.688,-66.422,-177.225,7.463,148.607
C08608=1173.760,260.440,-66.394,-177.227,7.460,148.607
C08609=1173.764,260.191,-66.367,-177.230,7.458,148.607
C08610=1173.769,259.943,-66.339,-177.232,7.455,148.607
C08611=1173.773,259.694,-66.312,-177.235,7.452,148.607
C08612=1173.778,259.446,-66.284,-177.238,7.449,148.607
C08613=1173.782,259.197,-66.257,-177.240,7.447,148.607
C08614=1173.786,258.949,-66.228,-177.243,7.444,148.608
C08615=1173.791,258.700,-66.201,-177.246,7.441,148.608
C08616=1173.795,258.452,-66.174,-177.248,7.439,148.608
C08617=1173.799,258.203,-66.146,-177.251,7.436,148.608
C08618=1173.803,257.955,-66.118,-177.254,7.433,148.608
C08619=1173.808,257.707,-66.091,-177.256,7.430,148.608
C08620=1173.812,257.458,-66.063,-177.259,7.428,148.608
C08621=1173.817,257.210,-66.036,-177.262,7.425,148.608
C08622=1173.821,256.961,-66.009,-177.264,7.422,148.608
C08623=1173.826,256.713,-65.981,-177.267,7.420,148.608
C08624=1173.830,256.464,-65.954,-177.269,7.417,148.608
C08625=1173.834,256.216,-65.927,-177.272,7.414,148.608
C08626=1173.839,255.968,-65.899,-177.275,7.413,148.609
C08627=1173.843,255.719,-65.872,-177.277,7.410,148.609
C08628=1173.847,255.470,-65.845,-177.280,7.407,148.609
C08629=1173.852,255.222,-65.817,-177.282,7.405,148.609
C08630=1173.856,254.974,-65.790,-177.285,7.402,148.609
C08631=1173.861,254.725,-65.763,-177.288,7.399,148.609
C08632=1173.865,254.477,-65.734,-177.291,7.397,148.609
C08633=1173.869,254.228,-65.707,-177.293,7.394,148.610
C08634=1173.874,253.980,-65.680,-177.296,7.391,148.610
C08635=1173.879,253.731,-65.653,-177.298,7.389,148.610
C08636=1173.883,253.483,-65.626,-177.301,7.386,148.610
C08637=1173.887,253.234,-65.598,-177.304,7.383,148.610
C08638=1173.892,252.986,-65.571,-177.306,7.381,148.610
C08639=1173.896,252.737,-65.545,-177.309,7.378,148.610
C08640=1173.900,252.489,-65.518,-177.312,7.375,148.610
C08641=1173.905,252.241,-65.490,-177.314,7.373,148.610
C08642=1173.909,251.992,-65.462,-177.317,7.370,148.611
C08643=1173.913,251.743,-65.435,-177.320,7.367,148.611
C08644=1173.918,251.495,-65.408,-177.322,7.365,148.611
C08645=1173.923,251.246,-65.381,-177.325,7.362,148.611
C08646=1173.927,250.998,-65.355,-177.328,7.359,148.611
C08647=1173.931,250.750,-65.328,-177.330,7.357,148.611
C08648=1173.936,250.501,-65.301,-177.333,7.354,148.611
C08649=1173.940,250.252,-65.273,-177.336,7.351,148.611
C08650=1173.945,250.003,-65.246,-177.338,7.349,148.611
C08651=1173.949,249.755,-65.220,-177.341,7.347,148.612
C08652=1173.953,249.507,-65.193,-177.344,7.344,148.612
C08653=1173.958,249.258,-65.165,-177.346,7.342,148.612
C08654=1173.963,249.010,-65.138,-177.349,7.339,148.612
C08655=1173.967,248.761,-65.111,-177.351,7.336,148.612
C08656=1173.971,248.513,-65.085,-177.354,7.334,148.612
C08657=1173.975,248.264,-65.057,-177.357,7.331,148.612
C08658=1173.980,248.015,-65.030,-177.359,7.329,148.612
C08659=1173.985,247.767,-65.003,-177.362,7.326,148.613
C08660=1173.988,247.519,-64.977,-177.365,7.323,148.613
C08661=1173.993,247.270,-64.950,-177.367,7.321,148.613
C08662=1173.998,247.022,-64.923,-177.370,7.318,148.613
C08663=1174.002,246.774,-64.896,-177.373,7.315,148.613
C08664=1174.006,246.525,-64.869,-177.375,7.313,148.613
C08665=1174.011,246.277,-64.842,-177.378,7.310,148.613
C08666=1174.015,246.028,-64.816,-177.380,7.308,148.614
C08667=1174.020,245.779,-64.789,-177.384,7.305,148.614
C08668=1174.025,245.531,-64.762,-177.386,7.303,148.614
C08669=1174.028,245.283,-64.736,-177.389,7.300,148.614
C08670=1174.033,245.034,-64.709,-177.391,7.297,148.614
C08671=1174.038,244.785,-64.682,-177.394,7.296,148.614
C08672=1174.042,244.537,-64.656,-177.397,7.293,148.614
C08673=1174.047,244.288,-64.629,-177.399,7.290,148.614
C08674=1174.051,244.040,-64.602,-177.402,7.288,148.615
C08675=1174.055,243.791,-64.576,-177.405,7.285,148.615
C08676=1174.060,243.542,-64.549,-177.407,7.283,148.615
C08677=1174.064,243.294,-64.523,-177.410,7.280,148.615
C08678=1174.069,243.046,-64.495,-177.413,7.277,148.615
C08679=1174.073,242.797,-64.470,-177.415,7.275,148.615
C08680=1174.078,242.549,-64.443,-177.418,7.272,148.615
C08681=1174.082,242.300,-64.416,-177.421,7.270,148.616
C08682=1174.086,242.051,-64.390,-177.423,7.267,148.616
C08683=1174.090,241.803,-64.363,-177.426,7.264,148.616
C08684=1174.095,241.555,-64.336,-177.429,7.263,148.616
C08685=1174.099,241.306,-64.311,-177.432,7.260,148.616
C08686=1174.104,241.057,-64.284,-177.434,7.257,148.616
C08687=1174.108,240.808,-64.258,-177.437,7.255,148.617
C08688=1174.113,240.560,-64.231,-177.439,7.253,148.617
C08689=1174.117,240.311,-64.205,-177.442,7.250,148.617
C08690=1174.122,240.063,-64.178,-177.445,7.247,148.617
C08691=1174.126,239.814,-64.152,-177.447,7.245,148.617
C08692=1174.131,239.565,-64.125,-177.450,7.242,148.617
C08693=1174.135,239.317,-64.099,-177.453,7.240,148.618
C08694=1174.139,239.068,-64.072,-177.455,7.237,148.618
C08695=1174.144,238.820,-64.047,-177.458,7.235,148.618
C08696=1174.149,238.571,-64.020,-177.461,7.232,148.618
C08697=1174.153,238.323,-63.994,-177.464,7.229,148.618
C08698=1174.157,238.074,-63.968,-177.466,7.227,148.618
C08699=1174.162,237.825,-63.941,-177.469,7.225,148.619
C08700=1174.166,237.577,-63.915,-177.471,7.223,148.619
C08701=1174.171,237.328,-63.888,-177.474,7.220,148.619
C08702=1174.175,237.080,-63.862,-177.477,7.218,148.619
C08703=1174.179,236.831,-63.836,-177.479,7.215,148.619
C08704=1174.185,236.560,-63.808,-177.483,7.212,148.619
C08705=1174.190,236.288,-63.779,-177.485,7.209,148.620
C08706=1174.194,236.016,-63.751,-177.488,7.207,148.620
C08707=1174.199,235.745,-63.722,-177.491,7.205,148.620
C08708=1174.204,235.496,-63.696,-177.494,7.202,148.620
C08709=1174.207,235.248,-63.670,-177.496,7.200,148.620
C08710=1174.212,234.999,-63.643,-177.499,7.197,148.621
C08711=1174.217,234.751,-63.618,-177.502,7.194,148.621
C08712=1174.221,234.502,-63.592,-177.504,7.192,148.621
C08713=1174.225,234.254,-63.566,-177.507,7.189,148.621
C08714=1174.230,234.004,-63.539,-177.510,7.187,148.621
C08715=1174.235,233.756,-63.514,-177.513,7.185,148.621
C08716=1174.239,233.508,-63.488,-177.515,7.182,148.622
C08717=1174.243,233.259,-63.462,-177.518,7.180,148.622
C08718=1174.248,233.010,-63.435,-177.520,7.178,148.622
C08719=1174.253,232.761,-63.410,-177.523,7.175,148.622
C08720=1174.257,232.513,-63.384,-177.526,7.173,148.622
C08721=1174.262,232.265,-63.358,-177.529,7.170,148.622
C08722=1174.267,232.015,-63.332,-177.531,7.168,148.623
C08723=1174.270,231.767,-63.306,-177.534,7.165,148.623
C08724=1174.275,231.518,-63.280,-177.536,7.163,148.623
C08725=1174.280,231.270,-63.255,-177.539,7.160,148.623
C08726=1174.284,231.022,-63.229,-177.542,7.158,148.623
C08727=1174.288,230.773,-63.203,-177.545,7.156,148.624
C08728=1174.293,230.524,-63.177,-177.547,7.154,148.624
C08729=1174.298,230.275,-63.151,-177.550,7.151,148.624
C08730=1174.302,230.027,-63.126,-177.552,7.149,148.624
C08731=1174.306,229.778,-63.100,-177.555,7.146,148.624
C08732=1174.311,229.530,-63.074,-177.558,7.144,148.625
C08733=1174.315,229.281,-63.049,-177.561,7.141,148.625
C08734=1174.319,229.032,-63.023,-177.563,7.139,148.625
C08735=1174.324,228.783,-62.997,-177.566,7.136,148.625
C08736=1174.329,228.535,-62.971,-177.569,7.135,148.625
C08737=1174.333,228.286,-62.945,-177.571,7.132,148.625
C08738=1174.338,228.037,-62.920,-177.574,7.130,148.626
C08739=1174.343,227.789,-62.894,-177.577,7.127,148.626
C08740=1174.347,227.540,-62.869,-177.579,7.125,148.626
C08741=1174.351,227.292,-62.843,-177.582,7.122,148.626
C08742=1174.356,227.044,-62.817,-177.584,7.120,148.626
C08743=1174.360,226.795,-62.792,-177.588,7.117,148.627
C08744=1174.365,226.545,-62.767,-177.590,7.115,148.627
C08745=1174.369,226.297,-62.741,-177.593,7.113,148.627
C08746=1174.374,226.048,-62.715,-177.595,7.110,148.627
C08747=1174.378,225.800,-62.690,-177.598,7.108,148.628
C08748=1174.383,225.551,-62.664,-177.601,7.106,148.628
C08749=1174.387,225.303,-62.639,-177.604,7.103,148.628
C08750=1174.391,225.053,-62.614,-177.606,7.101,148.628
C08751=1174.396,224.805,-62.588,-177.609,7.099,148.628
C08752=1174.400,224.556,-62.562,-177.612,7.096,148.628
C08753=1174.405,224.308,-62.537,-177.614,7.094,148.629
C08754=1174.410,224.059,-62.512,-177.617,7.091,148.629
C08755=1174.414,223.810,-62.486,-177.620,7.090,148.629
C08756=1174.419,223.562,-62.461,-177.622,7.087,148.629
C08757=1174.423,223.313,-62.435,-177.625,7.085,148.630
C08758=1174.428,223.064,-62.410,-177.628,7.082,148.630
C08759=1174.432,222.816,-62.385,-177.630,7.080,148.630
C08760=1174.436,222.567,-62.360,-177.633,7.077,148.630
C08761=1174.441,222.318,-62.335,-177.636,7.075,148.630
C08762=1174.445,222.070,-62.309,-177.638,7.073,148.631
C08763=1174.450,221.821,-62.284,-177.641,7.071,148.631
C08764=1174.455,221.572,-62.259,-177.644,7.069,148.631
C08765=1174.459,221.324,-62.233,-177.647,7.066,148.631
C08766=1174.464,221.074,-62.208,-177.649,7.064,148.632
C08767=1174.468,220.827,-62.183,-177.652,7.061,148.632
C08768=1174.472,220.578,-62.158,-177.655,7.059,148.632
C08769=1174.477,220.328,-62.133,-177.657,7.057,148.632
C08770=1174.482,220.080,-62.107,-177.660,7.055,148.632
C08771=1174.486,219.831,-62.082,-177.662,7.052,148.633
C08772=1174.490,219.583,-62.057,-177.666,7.050,148.633
C08773=1174.495,219.334,-62.032,-177.668,7.048,148.633
C08774=1174.500,219.086,-62.007,-177.671,7.045,148.633
C08775=1174.504,218.836,-61.982,-177.673,7.043,148.633
C08776=1174.509,218.588,-61.957,-177.676,7.041,148.634
C08777=1174.513,218.339,-61.932,-177.679,7.039,148.634
C08778=1174.518,218.091,-61.907,-177.681,7.036,148.634
C08779=1174.522,217.841,-61.882,-177.684,7.034,148.634
C08780=1174.527,217.593,-61.856,-177.687,7.032,148.635
C08781=1174.531,217.344,-61.832,-177.689,7.030,148.635
C08782=1174.536,217.096,-61.807,-177.692,7.027,148.635
C08783=1174.540,216.847,-61.782,-177.695,7.025,148.635
C08784=1174.545,216.598,-61.757,-177.698,7.022,148.636
C08785=1174.549,216.350,-61.732,-177.700,7.020,148.636
C08786=1174.554,216.101,-61.707,-177.703,7.019,148.636
C08787=1174.558,215.852,-61.683,-177.706,7.016,148.636
C08788=1174.563,215.604,-61.657,-177.708,7.014,148.637
C08789=1174.568,215.355,-61.633,-177.711,7.011,148.637
C08790=1174.571,215.106,-61.608,-177.714,7.009,148.637
C08791=1174.576,214.858,-61.583,-177.716,7.007,148.637
C08792=1174.581,214.609,-61.558,-177.719,7.004,148.637
C08793=1174.585,214.360,-61.534,-177.722,7.003,148.638
C08794=1174.590,214.112,-61.508,-177.725,7.000,148.638
C08795=1174.595,213.862,-61.483,-177.727,6.998,148.638
C08796=1174.599,213.614,-61.459,-177.730,6.996,148.639
C08797=1174.604,213.365,-61.434,-177.733,6.993,148.639
C08798=1174.608,213.116,-61.410,-177.735,6.991,148.639
C08799=1174.613,212.868,-61.385,-177.737,6.989,148.639
C08800=1174.617,212.618,-61.360,-177.741,6.987,148.639
C08801=1174.622,212.370,-61.335,-177.743,6.985,148.640
C08802=1174.627,212.121,-61.311,-177.746,6.982,148.640
C08803=1174.631,211.872,-61.286,-177.749,6.980,148.640
C08804=1174.635,211.624,-61.261,-177.751,6.978,148.640
C08805=1174.640,211.376,-61.237,-177.754,6.975,148.641
C08806=1174.644,211.126,-61.212,-177.757,6.973,148.641
C08807=1174.649,210.878,-61.188,-177.759,6.971,148.641
C08808=1174.654,210.608,-61.161,-177.762,6.969,148.641
C08809=1174.658,210.337,-61.134,-177.766,6.966,148.642
C08810=1174.664,210.066,-61.108,-177.768,6.964,148.642
C08811=1174.669,209.796,-61.081,-177.771,6.961,148.642
C08812=1174.674,209.546,-61.056,-177.774,6.960,148.642
C08813=1174.678,209.298,-61.032,-177.777,6.957,148.643
C08814=1174.682,209.050,-61.008,-177.779,6.955,148.643
C08815=1174.687,208.800,-60.983,-177.782,6.953,148.643
C08816=1174.691,208.552,-60.959,-177.784,6.950,148.643
C08817=1174.696,208.303,-60.934,-177.787,6.948,148.644
C08818=1174.700,208.054,-60.910,-177.790,6.946,148.644
C08819=1174.705,207.805,-60.885,-177.793,6.944,148.644
C08820=1174.710,207.557,-60.861,-177.795,6.942,148.644
C08821=1174.715,207.308,-60.837,-177.798,6.940,148.645
C08822=1174.719,207.059,-60.812,-177.801,6.937,148.645
C08823=1174.723,206.811,-60.788,-177.803,6.935,148.645
C08824=1174.728,206.562,-60.763,-177.806,6.933,148.646
C08825=1174.733,206.313,-60.739,-177.809,6.930,148.646
C08826=1174.736,206.064,-60.715,-177.811,6.929,148.646
C08827=1174.741,205.816,-60.690,-177.814,6.927,148.646
C08828=1174.746,205.567,-60.667,-177.817,6.924,148.646
C08829=1174.751,205.318,-60.642,-177.820,6.922,148.647
C08830=1174.755,205.069,-60.618,-177.822,6.920,148.647
C08831=1174.759,204.820,-60.594,-177.825,6.917,148.647
C08832=1174.765,204.572,-60.569,-177.828,6.916,148.648
C08833=1174.769,204.323,-60.545,-177.830,6.914,148.648
C08834=1174.774,204.074,-60.521,-177.833,6.911,148.648
C08835=1174.777,203.825,-60.497,-177.836,6.909,148.648
C08836=1174.783,203.576,-60.472,-177.838,6.907,148.649
C08837=1174.787,203.328,-60.448,-177.841,6.904,148.649
C08838=1174.792,203.079,-60.425,-177.844,6.903,148.649
C08839=1174.797,202.830,-60.400,-177.847,6.901,148.649
C08840=1174.801,202.581,-60.376,-177.849,6.898,148.650
C08841=1174.805,202.333,-60.352,-177.852,6.896,148.650
C08842=1174.810,202.084,-60.328,-177.855,6.894,148.650
C08843=1174.815,201.835,-60.304,-177.857,6.892,148.650
C08844=1174.819,201.586,-60.280,-177.860,6.890,148.651
C08845=1174.824,201.337,-60.256,-177.863,6.888,148.651
C08846=1174.828,201.088,-60.232,-177.865,6.886,148.651
C08847=1174.832,200.839,-60.209,-177.868,6.883,148.651
C08848=1174.838,200.591,-60.184,-177.871,6.881,148.652
C08849=1174.842,200.342,-60.160,-177.873,6.879,148.652
C08850=1174.847,200.093,-60.136,-177.876,6.877,148.652
C08851=1174.851,199.845,-60.112,-177.879,6.875,148.653
C08852=1174.856,199.596,-60.089,-177.882,6.873,148.653
C08853=1174.860,199.347,-60.065,-177.884,6.871,148.653
C08854=1174.865,199.098,-60.040,-177.887,6.868,148.653
C08855=1174.869,198.849,-60.016,-177.890,6.866,148.654
C08856=1174.874,198.600,-59.992,-177.892,6.865,148.654
C08857=1174.878,198.351,-59.969,-177.895,6.863,148.654
C08858=1174.883,198.103,-59.945,-177.898,6.860,148.655
C08859=1174.888,197.854,-59.922,-177.900,6.858,148.655
C08860=1174.892,197.605,-59.898,-177.903,6.856,148.655
C08861=1174.897,197.356,-59.874,-177.905,6.854,148.655
C08862=1174.901,197.108,-59.850,-177.909,6.852,148.656
C08863=1174.906,196.859,-59.827,-177.911,6.850,148.656
C08864=1174.911,196.610,-59.803,-177.913,6.848,148.656
C08865=1174.915,196.361,-59.778,-177.917,6.845,148.657
C08866=1174.920,196.111,-59.755,-177.919,6.843,148.657
C08867=1174.924,195.863,-59.731,-177.922,6.842,148.657
C08868=1174.929,195.614,-59.708,-177.924,6.839,148.657
C08869=1174.934,195.365,-59.684,-177.927,6.837,148.658
C08870=1174.938,195.117,-59.660,-177.930,6.835,148.658
C08871=1174.943,194.868,-59.637,-177.933,6.833,148.658
C08872=1174.947,194.619,-59.613,-177.935,6.831,148.659
C08873=1174.952,194.370,-59.589,-177.938,6.829,148.659
C08874=1174.956,194.121,-59.566,-177.941,6.827,148.659
C08875=1174.961,193.872,-59.543,-177.944,6.825,148.660
C08876=1174.965,193.624,-59.519,-177.946,6.823,148.660
C08877=1174.970,193.375,-59.495,-177.949,6.820,148.660
C08878=1174.975,193.126,-59.472,-177.952,6.819,148.660
C08879=1174.980,192.877,-59.448,-177.954,6.817,148.661
C08880=1174.984,192.628,-59.424,-177.957,6.815,148.661
C08881=1174.989,192.379,-59.401,-177.959,6.813,148.661
C08882=1174.993,192.130,-59.378,-177.962,6.810,148.662
C08883=1174.997,191.881,-59.355,-177.965,6.808,148.662
C08884=1175.002,191.633,-59.331,-177.967,6.806,148.662
C08885=1175.006,191.384,-59.307,-177.970,6.805,148.662
C08886=1175.011,191.135,-59.284,-177.973,6.802,148.663
C08887=1175.016,190.887,-59.261,-177.976,6.800,148.663
C08888=1175.021,190.638,-59.238,-177.978,6.798,148.663
C08889=1175.026,190.388,-59.214,-177.981,6.796,148.664
C08890=1175.031,190.139,-59.191,-177.983,6.794,148.664
C08891=1175.035,189.891,-59.167,-177.987,6.792,148.664
C08892=1175.039,189.642,-59.144,-177.989,6.790,148.665
C08893=1175.044,189.393,-59.121,-177.992,6.788,148.665
C08894=1175.048,189.144,-59.098,-177.994,6.786,148.665
C08895=1175.053,188.895,-59.074,-177.997,6.784,148.665
C08896=1175.058,188.646,-59.051,-178.000,6.782,148.666
C08897=1175.062,188.397,-59.027,-178.003,6.780,148.666
C08898=1175.066,188.148,-59.005,-178.005,6.778,148.666
C08899=1175.072,187.900,-58.982,-178.008,6.776,148.667
C08900=1175.076,187.651,-58.958,-178.010,6.774,148.667
C08901=1175.081,187.402,-58.935,-178.014,6.772,148.667
C08902=1175.086,187.153,-58.912,-178.016,6.770,148.668
C08903=1175.090,186.904,-58.889,-178.019,6.768,148.668
C08904=1175.094,186.655,-58.865,-178.021,6.766,148.668
C08905=1175.099,186.406,-58.842,-178.024,6.764,148.668
C08906=1175.104,186.157,-58.819,-178.027,6.762,148.669
C08907=1175.108,185.909,-58.796,-178.030,6.760,148.669
C08908=1175.113,185.660,-58.773,-178.032,6.758,148.669
C08909=1175.118,185.411,-58.750,-178.035,6.756,148.670
C08910=1175.122,185.162,-58.727,-178.037,6.754,148.670
C08911=1175.127,184.913,-58.704,-178.041,6.752,148.670
C08912=1175.132,184.644,-58.678,-178.043,6.750,148.671
C08913=1175.136,184.374,-58.654,-178.046,6.748,148.671
C08914=1175.142,184.104,-58.629,-178.049,6.746,148.671
C08915=1175.147,183.835,-58.604,-178.052,6.744,148.672
C08916=1175.151,183.586,-58.581,-178.055,6.742,148.672
C08917=1175.156,183.338,-58.558,-178.057,6.739,148.672
C08918=1175.161,183.088,-58.536,-178.060,6.737,148.673
C08919=1175.165,182.839,-58.513,-178.063,6.736,148.673
C08920=1175.170,182.590,-58.489,-178.065,6.734,148.673
C08921=1175.175,182.341,-58.466,-178.068,6.732,148.674
C08922=1175.179,182.092,-58.444,-178.071,6.730,148.674
C08923=1175.184,181.843,-58.421,-178.074,6.727,148.674
C08924=1175.188,181.595,-58.398,-178.076,6.725,148.674
C08925=1175.193,181.346,-58.375,-178.079,6.724,148.675
C08926=1175.198,181.097,-58.353,-178.082,6.722,148.675
C08927=1175.202,180.848,-58.330,-178.084,6.720,148.676
C08928=1175.207,180.599,-58.307,-178.087,6.718,148.676
C08929=1175.211,180.350,-58.284,-178.090,6.717,148.676
C08930=1175.217,180.101,-58.261,-178.092,6.714,148.676
C08931=1175.221,179.853,-58.239,-178.095,6.712,148.677
C08932=1175.226,179.603,-58.216,-178.098,6.710,148.677
C08933=1175.230,179.354,-58.193,-178.100,6.708,148.677
C08934=1175.235,179.106,-58.170,-178.103,6.707,148.678
C08935=1175.239,178.857,-58.148,-178.106,6.705,148.678
C08936=1175.244,178.607,-58.125,-178.108,6.703,148.679
C08937=1175.248,178.358,-58.103,-178.112,6.700,148.679
C08938=1175.253,178.110,-58.080,-178.114,6.698,148.679
C08939=1175.257,177.861,-58.057,-178.117,6.697,148.679
C08940=1175.262,177.611,-58.034,-178.119,6.695,148.680
C08941=1175.267,177.363,-58.012,-178.122,6.693,148.680
C08942=1175.272,177.114,-57.989,-178.125,6.691,148.680
C08943=1175.276,176.865,-57.967,-178.127,6.689,148.681
C08944=1175.282,176.616,-57.944,-178.130,6.688,148.681
C08945=1175.286,176.367,-57.922,-178.133,6.685,148.682
C08946=1175.291,176.118,-57.899,-178.135,6.683,148.682
C08947=1175.295,175.870,-57.877,-178.138,6.681,148.682
C08948=1175.299,175.620,-57.855,-178.141,6.679,148.682
C08949=1175.304,175.371,-57.831,-178.143,6.678,148.683
C08950=1175.309,175.123,-57.809,-178.146,6.676,148.683
C08951=1175.314,174.873,-57.787,-178.149,6.674,148.683
C08952=1175.318,174.624,-57.764,-178.151,6.672,148.684
C08953=1175.323,174.376,-57.742,-178.154,6.671,148.684
C08954=1175.327,174.127,-57.719,-178.157,6.668,148.685
C08955=1175.332,173.878,-57.697,-178.160,6.666,148.685
C08956=1175.337,173.629,-57.675,-178.162,6.664,148.685
C08957=1175.341,173.380,-57.652,-178.165,6.662,148.685
C08958=1175.346,173.131,-57.630,-178.168,6.661,148.686
C08959=1175.350,172.882,-57.608,-178.170,6.659,148.686
C08960=1175.356,172.633,-57.585,-178.173,6.657,148.687
C08961=1175.360,172.384,-57.563,-178.176,6.655,148.687
C08962=1175.364,172.135,-57.541,-178.178,6.654,148.687
C08963=1175.370,171.886,-57.518,-178.181,6.652,148.688
C08964=1175.374,171.637,-57.496,-178.184,6.650,148.688
C08965=1175.379,171.388,-57.474,-178.187,6.647,148.688
C08966=1175.384,171.139,-57.452,-178.190,6.646,148.689
C08967=1175.388,170.891,-57.429,-178.192,6.644,148.689
C08968=1175.393,170.641,-57.407,-178.195,6.642,148.689
C08969=1175.397,170.392,-57.385,-178.197,6.640,148.690
C08970=1175.402,170.143,-57.363,-178.200,6.638,148.690
C08971=1175.406,169.894,-57.340,-178.203,6.636,148.690
C08972=1175.411,169.646,-57.319,-178.205,6.635,148.691
C08973=1175.416,169.396,-57.296,-178.208,6.633,148.691
C08974=1175.421,169.147,-57.274,-178.211,6.631,148.691
C08975=1175.425,168.898,-57.252,-178.213,6.629,148.692
C08976=1175.430,168.649,-57.230,-178.216,6.628,148.692
C08977=1175.435,168.400,-57.208,-178.219,6.626,148.693
C08978=1175.439,168.152,-57.186,-178.221,6.624,148.693
C08979=1175.444,167.902,-57.163,-178.225,6.622,148.693
C08980=1175.449,167.654,-57.142,-178.227,6.620,148.694
C08981=1175.453,167.404,-57.120,-178.230,6.618,148.694
C08982=1175.458,167.156,-57.098,-178.233,6.616,148.694
C08983=1175.462,166.906,-57.076,-178.235,6.614,148.695
C08984=1175.468,166.657,-57.054,-178.238,6.612,148.695
C08985=1175.472,166.408,-57.032,-178.240,6.611,148.695
C08986=1175.477,166.159,-57.010,-178.243,6.609,148.696
C08987=1175.481,165.910,-56.988,-178.246,6.607,148.696
C08988=1175.486,165.662,-56.966,-178.248,6.605,148.696
C08989=1175.491,165.412,-56.944,-178.251,6.604,148.697
C08990=1175.495,165.164,-56.922,-178.254,6.602,148.697
C08991=1175.500,164.915,-56.901,-178.256,6.600,148.697
C08992=1175.505,164.666,-56.879,-178.259,6.598,148.698
C08993=1175.509,164.417,-56.857,-178.262,6.596,148.698
C08994=1175.514,164.168,-56.835,-178.264,6.595,148.699
C08995=1175.519,163.919,-56.813,-178.267,6.593,148.699
C08996=1175.524,163.669,-56.791,-178.270,6.591,148.699
C08997=1175.528,163.421,-56.769,-178.273,6.589,148.700
C08998=1175.533,163.172,-56.747,-178.275,6.588,148.700
C08999=1175.538,162.923,-56.725,-178.278,6.586,148.700
C09000=1175.543,162.673,-56.704,-178.281,6.584,148.701
C09001=1175.547,162.424,-56.682,-178.283,6.582,148.701
C09002=1175.552,162.175,-56.661,-178.286,6.581,148.702
C09003=1175.557,161.927,-56.639,-178.289,6.579,148.702
C09004=1175.561,161.677,-56.617,-178.291,6.577,148.702
C09005=1175.566,161.429,-56.595,-178.294,6.575,148.703
C09006=1175.570,161.179,-56.574,-178.297,6.574,148.703
C09007=1175.575,160.930,-56.552,-178.299,6.572,148.703
C09008=1175.580,160.682,-56.530,-178.302,6.570,148.704
C09009=1175.584,160.432,-56.508,-178.305,6.568,148.704
C09010=1175.589,160.184,-56.487,-178.307,6.567,148.705
C09011=1175.594,159.935,-56.466,-178.310,6.565,148.705
C09012=1175.598,159.685,-56.444,-178.313,6.563,148.705
C09013=1175.603,159.437,-56.423,-178.316,6.561,148.706
C09014=1175.608,159.188,-56.401,-178.318,6.559,148.706
C09015=1175.612,158.938,-56.380,-178.321,6.558,148.706
C09016=1175.618,158.669,-56.356,-178.324,6.555,148.707
C09017=1175.622,158.400,-56.333,-178.327,6.553,148.707
C09018=1175.628,158.131,-56.309,-178.330,6.552,148.708
C09019=1175.633,157.863,-56.287,-178.333,6.550,148.708
C09020=1175.637,157.613,-56.265,-178.335,6.548,148.708
C09021=1175.642,157.365,-56.243,-178.338,6.547,148.709
C09022=1175.647,157.115,-56.222,-178.341,6.545,148.709
C09023=1175.652,156.866,-56.200,-178.343,6.543,148.710
C09024=1175.656,156.617,-56.180,-178.346,6.541,148.710
C09025=1175.661,156.368,-56.158,-178.349,6.540,148.710
C09026=1175.665,156.119,-56.136,-178.352,6.538,148.711
C09027=1175.670,155.870,-56.115,-178.354,6.536,148.711
C09028=1175.675,155.621,-56.094,-178.357,6.534,148.711
C09029=1175.680,155.372,-56.073,-178.360,6.533,148.712
C09030=1175.684,155.123,-56.051,-178.362,6.531,148.712
C09031=1175.689,154.874,-56.030,-178.365,6.529,148.713
C09032=1175.694,154.625,-56.008,-178.368,6.527,148.713
C09033=1175.699,154.376,-55.987,-178.370,6.526,148.713
C09034=1175.703,154.127,-55.966,-178.373,6.524,148.714
C09035=1175.708,153.877,-55.945,-178.376,6.522,148.714
C09036=1175.713,153.629,-55.923,-178.378,6.520,148.714
C09037=1175.718,153.379,-55.902,-178.381,6.519,148.715
C09038=1175.722,153.131,-55.881,-178.384,6.517,148.715
C09039=1175.727,152.881,-55.860,-178.386,6.515,148.716
C09040=1175.732,152.633,-55.838,-178.389,6.513,148.716
C09041=1175.737,152.383,-55.817,-178.392,6.512,148.717
C09042=1175.741,152.134,-55.797,-178.395,6.510,148.717
C09043=1175.746,151.886,-55.775,-178.398,6.508,148.717
C09044=1175.751,151.636,-55.754,-178.400,6.507,148.718
C09045=1175.755,151.387,-55.733,-178.403,6.506,148.718
C09046=1175.760,151.138,-55.712,-178.405,6.504,148.718
C09047=1175.765,150.889,-55.691,-178.408,6.502,148.719
C09048=1175.770,150.640,-55.669,-178.411,6.500,148.719
C09049=1175.774,150.391,-55.649,-178.413,6.499,148.720
C09050=1175.779,150.141,-55.628,-178.416,6.497,148.720
C09051=1175.783,149.893,-55.606,-178.419,6.495,148.720
C09052=1175.788,149.644,-55.585,-178.421,6.493,148.721
C09053=1175.793,149.394,-55.565,-178.424,6.492,148.721
C09054=1175.798,149.146,-55.543,-178.427,6.490,148.722
C09055=1175.803,148.897,-55.522,-178.429,6.488,148.722
C09056=1175.807,148.647,-55.501,-178.433,6.487,148.723
C09057=1175.812,148.398,-55.481,-178.435,6.485,148.723
C09058=1175.817,148.149,-55.459,-178.437,6.484,148.723
C09059=1175.821,147.900,-55.439,-178.440,6.482,148.724
C09060=1175.826,147.651,-55.418,-178.443,6.481,148.724
C09061=1175.831,147.402,-55.397,-178.446,6.479,148.724
C09062=1175.836,147.153,-55.376,-178.448,6.477,148.725
C09063=1175.841,146.904,-55.355,-178.451,6.475,148.725
C09064=1175.845,146.655,-55.334,-178.454,6.474,148.726
C09065=1175.850,146.405,-55.313,-178.456,6.472,148.726
C09066=1175.854,146.156,-55.293,-178.459,6.470,148.726
C09067=1175.859,145.907,-55.272,-178.462,6.469,148.727
C09068=1175.864,145.658,-55.251,-178.465,6.467,148.727
C09069=1175.869,145.409,-55.230,-178.467,6.466,148.728
C09070=1175.873,145.160,-55.210,-178.470,6.464,148.728
C09071=1175.878,144.911,-55.188,-178.472,6.462,148.728
C09072=1175.883,144.662,-55.168,-178.475,6.461,148.729
C09073=1175.888,144.413,-55.147,-178.478,6.459,148.729
C09074=1175.892,144.164,-55.127,-178.480,6.457,148.730
C09075=1175.897,143.915,-55.106,-178.483,6.455,148.730
C09076=1175.902,143.666,-55.085,-178.486,6.454,148.731
C09077=1175.907,143.417,-55.064,-178.489,6.452,148.731
C09078=1175.912,143.168,-55.044,-178.492,6.451,148.731
C09079=1175.915,142.918,-55.023,-178.494,6.450,148.732
C09080=1175.921,142.669,-55.002,-178.497,6.448,148.732
C09081=1175.925,142.420,-54.982,-178.499,6.446,148.733
C09082=1175.930,142.171,-54.961,-178.502,6.444,148.733
C09083=1175.935,141.922,-54.940,-178.505,6.443,148.733
C09084=1175.940,141.672,-54.920,-178.507,6.441,148.734
C09085=1175.944,141.424,-54.899,-178.510,6.439,148.734
C09086=1175.949,141.175,-54.879,-178.513,6.438,148.735
C09087=1175.954,140.925,-54.858,-178.515,6.437,148.735
C09088=1175.958,140.676,-54.837,-178.518,6.435,148.736
C09089=1175.963,140.427,-54.818,-178.521,6.433,148.736
C09090=1175.968,140.178,-54.797,-178.523,6.432,148.736
C09091=1175.973,139.929,-54.776,-178.526,6.430,148.737
C09092=1175.977,139.680,-54.756,-178.529,6.428,148.737
C09093=1175.983,139.431,-54.735,-178.532,6.427,148.738
C09094=1175.987,139.182,-54.715,-178.534,6.426,148.738
C09095=1175.992,138.933,-54.695,-178.537,6.424,148.738
C09096=1175.997,138.683,-54.674,-178.539,6.422,148.739
C09097=1176.002,138.434,-54.654,-178.542,6.420,148.739
C09098=1176.006,138.185,-54.634,-178.545,6.419,148.740
C09099=1176.011,137.936,-54.613,-178.548,6.417,148.740
C09100=1176.016,137.687,-54.592,-178.551,6.416,148.741
C09101=1176.020,137.438,-54.573,-178.553,6.415,148.741
C09102=1176.025,137.189,-54.552,-178.556,6.413,148.741
C09103=1176.030,136.939,-54.531,-178.558,6.411,148.742
C09104=1176.034,136.690,-54.511,-178.561,6.409,148.742
C09105=1176.039,136.441,-54.491,-178.564,6.408,148.743
C09106=1176.044,136.192,-54.471,-178.567,6.406,148.743
C09107=1176.049,135.943,-54.450,-178.569,6.405,148.744
C09108=1176.054,135.694,-54.430,-178.572,6.404,148.744
C09109=1176.059,135.445,-54.410,-178.574,6.402,148.744
C09110=1176.063,135.196,-54.390,-178.577,6.400,148.745
C09111=1176.068,134.947,-54.369,-178.580,6.398,148.745
C09112=1176.073,134.697,-54.349,-178.583,6.397,148.746
C09113=1176.077,134.448,-54.329,-178.585,6.396,148.746
C09114=1176.082,134.199,-54.309,-178.588,6.394,148.747
C09115=1176.087,133.950,-54.289,-178.590,6.393,148.747
C09116=1176.092,133.701,-54.269,-178.593,6.391,148.747
C09117=1176.097,133.452,-54.249,-178.596,6.389,148.748
C09118=1176.102,133.203,-54.228,-178.598,6.389,148.748
C09119=1176.106,132.953,-54.209,-178.601,6.387,148.749
C09120=1176.111,132.685,-54.187,-178.604,6.385,148.749
C09121=1176.117,132.416,-54.165,-178.607,6.384,148.750
C09122=1176.121,132.148,-54.143,-178.610,6.382,148.750
C09123=1176.127,131.879,-54.122,-178.612,6.380,148.751
C09124=1176.132,131.629,-54.102,-178.616,6.379,148.751
C09125=1176.136,131.380,-54.082,-178.618,6.377,148.752
C09126=1176.141,131.132,-54.062,-178.621,6.375,148.752
C09127=1176.146,130.883,-54.042,-178.624,6.374,148.752
C09128=1176.150,130.633,-54.022,-178.626,6.373,148.753
C09129=1176.155,130.384,-54.002,-178.629,6.371,148.753
C09130=1176.160,130.134,-53.982,-178.632,6.369,148.754
C09131=1176.165,129.886,-53.962,-178.634,6.368,148.754
C09132=1176.170,129.636,-53.942,-178.637,6.366,148.755
C09133=1176.175,129.388,-53.922,-178.639,6.365,148.755
C09134=1176.179,129.138,-53.902,-178.642,6.363,148.755
C09135=1176.184,128.890,-53.882,-178.645,6.362,148.756
C09136=1176.189,128.640,-53.862,-178.648,6.360,148.756
C09137=1176.194,128.391,-53.843,-178.651,6.358,148.757
C09138=1176.198,128.142,-53.822,-178.653,6.358,148.757
C09139=1176.203,127.892,-53.803,-178.656,6.356,148.758
C09140=1176.208,127.643,-53.783,-178.659,6.354,148.758
C09141=1176.213,127.394,-53.763,-178.661,6.353,148.759
C09142=1176.218,127.145,-53.743,-178.663,6.352,148.759
C09143=1176.222,126.895,-53.724,-178.666,6.350,148.759
